LIN {X 0.102,Y -450.857,Z 437.939,A 0.000,B 0.000,C 90.000,E1 204.975} C_DIS
LIN {X -0.124,Y -447.406,Z 437.930,A 0.000,B 0.000,C 90.000,E1 203.387} C_DIS
LIN {X -0.058,Y -442.632,Z 437.917,A 0.000,B 0.000,C 90.000,E1 201.099} C_DIS
LIN {X -0.035,Y -437.484,Z 437.903,A 0.000,B 0.000,C 90.000,E1 198.471} C_DIS
LIN {X 0.091,Y -434.534,Z 437.893,A 0.000,B 0.000,C 90.000,E1 196.804} C_DIS
LIN {X 0.077,Y -430.659,Z 437.881,A 0.000,B 0.000,C 90.000,E1 194.481} C_DIS
LIN {X -0.065,Y -426.530,Z 437.866,A 0.000,B 0.000,C 90.000,E1 191.827} C_DIS
LIN {X -0.012,Y -422.037,Z 437.847,A 0.000,B 0.000,C 90.000,E1 188.454} C_DIS
LIN {X -0.048,Y -419.643,Z 437.836,A 0.000,B 0.000,C 90.000,E1 186.429} C_DIS
LIN {X 0.164,Y -417.753,Z 437.826,A 0.000,B 0.000,C 90.000,E1 184.702} C_DIS
LIN {X -0.025,Y -414.692,Z 437.807,A 0.000,B 0.000,C 90.000,E1 181.318} C_DIS
LIN {X 0.048,Y -412.866,Z 437.792,A 0.000,B 0.000,C 90.000,E1 178.568} C_DIS
LIN {X 0.133,Y -411.529,Z 437.773,A 0.000,B 0.000,C 90.000,E1 175.122} C_DIS
LIN {X -0.070,Y -411.506,Z 437.748,A 0.000,B 0.000,C 90.000,E1 170.679} C_DIS
LIN {X -0.129,Y -412.288,Z 437.733,A 0.000,B 0.000,C 90.000,E1 167.937} C_DIS
LIN {X -0.220,Y -414.218,Z 437.714,A 0.000,B 0.000,C 90.000,E1 164.519} C_DIS
LIN {X 0.137,Y -417.750,Z 437.691,A 0.000,B 0.000,C 90.000,E1 160.369} C_DIS
LIN {X -0.098,Y -422.139,Z 437.670,A 0.000,B 0.000,C 90.000,E1 156.666} C_DIS
LIN {X 0.070,Y -425.355,Z 437.657,A 0.000,B 0.000,C 90.000,E1 154.280} C_DIS
LIN {X 0.108,Y -429.539,Z 437.642,A 0.000,B 0.000,C 90.000,E1 151.591} C_DIS
LIN {X -0.093,Y -432.946,Z 437.631,A 0.000,B 0.000,C 90.000,E1 149.616} C_DIS
LIN {X 0.262,Y -437.222,Z 437.618,A 0.000,B 0.000,C 90.000,E1 147.248} C_DIS
LIN {X -0.031,Y -441.130,Z 437.607,A 0.000,B 0.000,C 90.000,E1 145.308} C_DIS
LIN {X 0.081,Y -447.445,Z 437.591,A 0.000,B 0.000,C 90.000,E1 142.351} C_DIS
LIN {X 0.182,Y -453.544,Z 437.577,A 0.000,B 0.000,C 90.000,E1 139.747} C_DIS
LIN {X 0.005,Y -457.461,Z 437.568,A 0.000,B 0.000,C 90.000,E1 138.162} C_DIS
LIN {X 0.201,Y -461.161,Z 437.559,A 0.000,B 0.000,C 90.000,E1 136.539} C_DIS
LIN {X 0.021,Y -463.308,Z 437.553,A 0.000,B 0.000,C 90.000,E1 135.607} C_DIS
LIN {X -0.141,Y -465.220,Z 437.548,A 0.000,B 0.000,C 90.000,E1 134.676} C_DIS
LIN {X -0.015,Y -466.473,Z 437.545,A 0.000,B 0.000,C 90.000,E1 134.028} C_DIS
LIN {X -0.059,Y -468.597,Z 437.538,A 0.000,B 0.000,C 90.000,E1 132.771} C_DIS
LIN {X -0.151,Y -469.844,Z 437.532,A 0.000,B 0.000,C 90.000,E1 131.838} C_DIS
LIN {X 0.125,Y -470.762,Z 437.527,A 0.000,B 0.000,C 90.000,E1 130.862} C_DIS
LIN {X -0.025,Y -471.260,Z 437.524,A 0.000,B 0.000,C 90.000,E1 130.253} C_DIS
LIN {X -0.096,Y -471.592,Z 437.518,A 0.000,B 0.000,C 90.000,E1 129.322} C_DIS
LIN {X -0.101,Y -471.281,Z 437.513,A 0.000,B 0.000,C 90.000,E1 128.382} C_DIS
LIN {X -0.106,Y -470.509,Z 437.508,A 0.000,B 0.000,C 90.000,E1 127.443} C_DIS
LIN {X -0.119,Y -469.371,Z 437.503,A 0.000,B 0.000,C 90.000,E1 126.503} C_DIS
LIN {X 0.230,Y -467.871,Z 437.498,A 0.000,B 0.000,C 90.000,E1 125.518} C_DIS
LIN {X -0.089,Y -465.949,Z 437.492,A 0.000,B 0.000,C 90.000,E1 124.612} C_DIS
LIN {X -0.041,Y -463.642,Z 437.487,A 0.000,B 0.000,C 90.000,E1 123.658} C_DIS
LIN {X -0.150,Y -461.927,Z 437.483,A 0.000,B 0.000,C 90.000,E1 123.038} C_DIS
LIN {X -0.021,Y -458.176,Z 437.476,A 0.000,B 0.000,C 90.000,E1 121.750} C_DIS
LIN {X 0.043,Y -453.962,Z 437.469,A 0.000,B 0.000,C 90.000,E1 120.463} C_DIS
LIN {X 0.112,Y -450.602,Z 437.464,A 0.000,B 0.000,C 90.000,E1 119.489} C_DIS
LIN {X -0.105,Y -444.709,Z 437.455,A 0.000,B 0.000,C 90.000,E1 117.897} C_DIS
LIN {X -0.140,Y -439.938,Z 437.448,A 0.000,B 0.000,C 90.000,E1 116.616} C_DIS
LIN {X -0.180,Y -439.926,Z 437.448,A 0.000,B 0.000,C 90.000,E1 116.616} C_DIS
LIN {X -0.108,Y -444.759,Z 437.439,A 0.000,B 0.000,C 90.000,E1 114.951} C_DIS
LIN {X -0.138,Y -454.729,Z 437.415,A 0.000,B 0.000,C 90.000,E1 110.737} C_DIS
LIN {X -0.015,Y -457.367,Z 437.410,A 0.000,B 0.000,C 90.000,E1 109.758} C_DIS
LIN {X 0.070,Y -465.999,Z 437.387,A 0.000,B 0.000,C 90.000,E1 105.607} C_DIS
LIN {X -0.207,Y -467.566,Z 437.383,A 0.000,B 0.000,C 90.000,E1 105.009} C_DIS
LIN {X -0.024,Y -468.575,Z 437.380,A 0.000,B 0.000,C 90.000,E1 104.356} C_DIS
LIN {X 0.203,Y -475.799,Z 437.357,A 0.000,B 0.000,C 90.000,E1 100.254} C_DIS
LIN {X 0.041,Y -476.304,Z 437.355,A 0.000,B 0.000,C 90.000,E1 99.962} C_DIS
LIN {X -0.012,Y -481.788,Z 437.331,A 0.000,B 0.000,C 90.000,E1 95.625} C_DIS
LIN {X -0.165,Y -482.171,Z 437.330,A 0.000,B 0.000,C 90.000,E1 95.334} C_DIS
LIN {X -0.235,Y -485.307,Z 437.306,A 0.000,B 0.000,C 90.000,E1 91.031} C_DIS
LIN {X 0.074,Y -485.537,Z 437.304,A 0.000,B 0.000,C 90.000,E1 90.688} C_DIS
LIN {X -0.204,Y -486.319,Z 437.282,A 0.000,B 0.000,C 90.000,E1 86.731} C_DIS
LIN {X -0.069,Y -486.306,Z 437.278,A 0.000,B 0.000,C 90.000,E1 86.102} C_DIS
LIN {X 0.136,Y -484.695,Z 437.254,A 0.000,B 0.000,C 90.000,E1 81.781} C_DIS
LIN {X 0.004,Y -484.601,Z 437.253,A 0.000,B 0.000,C 90.000,E1 81.489} C_DIS
LIN {X -0.116,Y -480.535,Z 437.227,A 0.000,B 0.000,C 90.000,E1 76.881} C_DIS
LIN {X 0.248,Y -474.286,Z 437.201,A 0.000,B 0.000,C 90.000,E1 72.181} C_DIS
LIN {X 0.067,Y -473.850,Z 437.199,A 0.000,B 0.000,C 90.000,E1 71.891} C_DIS
LIN {X 0.175,Y -466.257,Z 437.175,A 0.000,B 0.000,C 90.000,E1 67.486} C_DIS
LIN {X 0.118,Y -465.828,Z 437.173,A 0.000,B 0.000,C 90.000,E1 67.177} C_DIS
LIN {X 0.057,Y -465.235,Z 437.172,A 0.000,B 0.000,C 90.000,E1 66.869} C_DIS
LIN {X -0.019,Y -463.619,Z 437.168,A 0.000,B 0.000,C 90.000,E1 66.177} C_DIS
LIN {X -0.059,Y -463.611,Z 437.168,A 0.000,B 0.000,C 90.000,E1 66.177} C_DIS
LIN {X 0.020,Y -474.649,Z 437.159,A 0.000,B 0.000,C 90.000,E1 64.665} C_DIS
LIN {X -0.068,Y -483.723,Z 437.152,A 0.000,B 0.000,C 90.000,E1 63.435} C_DIS
LIN {X 0.143,Y -487.056,Z 437.150,A 0.000,B 0.000,C 90.000,E1 62.948} C_DIS
LIN {X -0.053,Y -491.221,Z 437.146,A 0.000,B 0.000,C 90.000,E1 62.359} C_DIS
LIN {X 0.047,Y -497.047,Z 437.141,A 0.000,B 0.000,C 90.000,E1 61.435} C_DIS
LIN {X 0.169,Y -501.422,Z 437.137,A 0.000,B 0.000,C 90.000,E1 60.667} C_DIS
LIN {X 0.142,Y -505.295,Z 437.133,A 0.000,B 0.000,C 90.000,E1 59.921} C_DIS
LIN {X 0.082,Y -508.046,Z 437.130,A 0.000,B 0.000,C 90.000,E1 59.331} C_DIS
LIN {X 0.223,Y -509.913,Z 437.127,A 0.000,B 0.000,C 90.000,E1 58.869} C_DIS
LIN {X -0.246,Y -512.107,Z 437.124,A 0.000,B 0.000,C 90.000,E1 58.329} C_DIS
LIN {X 0.095,Y -513.096,Z 437.122,A 0.000,B 0.000,C 90.000,E1 57.995} C_DIS
LIN {X 0.079,Y -514.790,Z 437.119,A 0.000,B 0.000,C 90.000,E1 57.406} C_DIS
LIN {X -0.153,Y -516.775,Z 437.114,A 0.000,B 0.000,C 90.000,E1 56.548} C_DIS
LIN {X 0.141,Y -517.817,Z 437.111,A 0.000,B 0.000,C 90.000,E1 55.928} C_DIS
LIN {X 0.086,Y -518.891,Z 437.106,A 0.000,B 0.000,C 90.000,E1 55.055} C_DIS
LIN {X -0.087,Y -519.451,Z 437.101,A 0.000,B 0.000,C 90.000,E1 54.196} C_DIS
LIN {X 0.165,Y -519.607,Z 437.096,A 0.000,B 0.000,C 90.000,E1 53.290} C_DIS
LIN {X 0.000,Y -519.588,Z 437.091,A 0.000,B 0.000,C 90.000,E1 52.431} C_DIS
LIN {X 0.153,Y -519.326,Z 437.086,A 0.000,B 0.000,C 90.000,E1 51.537} C_DIS
LIN {X 0.251,Y -518.494,Z 437.080,A 0.000,B 0.000,C 90.000,E1 50.356} C_DIS
LIN {X -0.059,Y -517.555,Z 437.073,A 0.000,B 0.000,C 90.000,E1 49.218} C_DIS
LIN {X 0.003,Y -516.367,Z 437.067,A 0.000,B 0.000,C 90.000,E1 48.038} C_DIS
LIN {X -0.106,Y -514.780,Z 437.059,A 0.000,B 0.000,C 90.000,E1 46.581} C_DIS
LIN {X -0.276,Y -511.804,Z 437.044,A 0.000,B 0.000,C 90.000,E1 43.947} C_DIS
LIN {X -0.091,Y -510.209,Z 437.036,A 0.000,B 0.000,C 90.000,E1 42.447} C_DIS
LIN {X 0.200,Y -509.021,Z 437.029,A 0.000,B 0.000,C 90.000,E1 41.229} C_DIS
LIN {X -0.101,Y -506.220,Z 437.014,A 0.000,B 0.000,C 90.000,E1 38.588} C_DIS
LIN {X 0.091,Y -504.707,Z 437.006,A 0.000,B 0.000,C 90.000,E1 37.076} C_DIS
LIN {X 0.176,Y -503.686,Z 437.001,A 0.000,B 0.000,C 90.000,E1 36.171} C_DIS
LIN {X 0.029,Y -501.970,Z 436.993,A 0.000,B 0.000,C 90.000,E1 34.692} C_DIS
LIN {X 0.259,Y -500.091,Z 436.984,A 0.000,B 0.000,C 90.000,E1 33.166} C_DIS
LIN {X 0.064,Y -497.370,Z 436.973,A 0.000,B 0.000,C 90.000,E1 31.082} C_DIS
LIN {X -0.078,Y -495.355,Z 436.964,A 0.000,B 0.000,C 90.000,E1 29.589} C_DIS
LIN {X 0.228,Y -492.204,Z 436.951,A 0.000,B 0.000,C 90.000,E1 27.129} C_DIS
LIN {X 0.267,Y -488.755,Z 436.934,A 0.000,B 0.000,C 90.000,E1 24.079} C_DIS
LIN {X 0.006,Y -486.549,Z 436.920,A 0.000,B 0.000,C 90.000,E1 21.663} C_DIS
LIN {X 0.105,Y -485.254,Z 436.910,A 0.000,B 0.000,C 90.000,E1 19.812} C_DIS
LIN {X -0.156,Y -483.886,Z 436.898,A 0.000,B 0.000,C 90.000,E1 17.692} C_DIS
LIN {X 0.158,Y -483.262,Z 436.893,A 0.000,B 0.000,C 90.000,E1 16.732} C_DIS
LIN {X 0.036,Y -481.976,Z 436.883,A 0.000,B 0.000,C 90.000,E1 14.898} C_DIS
LIN {X 0.223,Y -480.003,Z 436.864,A 0.000,B 0.000,C 90.000,E1 11.478} C_DIS
LIN {X -0.002,Y -479.129,Z 436.850,A 0.000,B 0.000,C 90.000,E1 9.029} C_DIS
LIN {X -0.150,Y -478.666,Z 436.835,A 0.000,B 0.000,C 90.000,E1 6.258} C_DIS
LIN {X -0.195,Y -478.900,Z 436.821,A 0.000,B 0.000,C 90.000,E1 3.784} C_DIS
LIN {X -0.110,Y -480.493,Z 436.800,A 0.000,B 0.000,C 90.000,E1 0.057} C_DIS
LIN {X -0.097,Y -481.532,Z 436.792,A 0.000,B 0.000,C 90.000,E1 358.568} C_DIS
LIN {X -0.057,Y -483.080,Z 436.783,A 0.000,B 0.000,C 90.000,E1 357.020} C_DIS
LIN {X -0.092,Y -487.702,Z 436.763,A 0.000,B 0.000,C 90.000,E1 353.337} C_DIS
LIN {X -0.004,Y -492.402,Z 436.746,A 0.000,B 0.000,C 90.000,E1 350.274} C_DIS
LIN {X 0.038,Y -498.428,Z 436.728,A 0.000,B 0.000,C 90.000,E1 346.937} C_DIS
LIN {X 0.083,Y -505.796,Z 436.709,A 0.000,B 0.000,C 90.000,E1 343.630} C_DIS
LIN {X -0.024,Y -512.499,Z 436.694,A 0.000,B 0.000,C 90.000,E1 340.967} C_DIS
LIN {X 0.004,Y -518.050,Z 436.683,A 0.000,B 0.000,C 90.000,E1 338.901} C_DIS
LIN {X -0.086,Y -522.817,Z 436.673,A 0.000,B 0.000,C 90.000,E1 337.155} C_DIS
LIN {X 0.245,Y -526.906,Z 436.665,A 0.000,B 0.000,C 90.000,E1 335.665} C_DIS
LIN {X 0.275,Y -532.592,Z 436.654,A 0.000,B 0.000,C 90.000,E1 333.640} C_DIS
LIN {X 0.207,Y -538.348,Z 436.643,A 0.000,B 0.000,C 90.000,E1 331.641} C_DIS
LIN {X 0.058,Y -543.469,Z 436.633,A 0.000,B 0.000,C 90.000,E1 329.950} C_DIS
LIN {X 0.065,Y -547.624,Z 436.625,A 0.000,B 0.000,C 90.000,E1 328.535} C_DIS
LIN {X 0.103,Y -550.994,Z 436.619,A 0.000,B 0.000,C 90.000,E1 327.406} C_DIS
LIN {X -0.013,Y -557.487,Z 436.607,A 0.000,B 0.000,C 90.000,E1 325.182} C_DIS
LIN {X 0.186,Y -562.446,Z 436.597,A 0.000,B 0.000,C 90.000,E1 323.497} C_DIS
LIN {X 0.266,Y -566.630,Z 436.590,A 0.000,B 0.000,C 90.000,E1 322.110} C_DIS
LIN {X 0.381,Y -573.652,Z 436.578,A 0.000,B 0.000,C 90.000,E1 319.908} C_DIS
LIN {X 0.078,Y -579.838,Z 436.567,A 0.000,B 0.000,C 90.000,E1 318.038} C_DIS
LIN {X -0.301,Y -584.991,Z 436.558,A 0.000,B 0.000,C 90.000,E1 316.458} C_DIS
LIN {X 0.089,Y -589.319,Z 436.551,A 0.000,B 0.000,C 90.000,E1 315.081} C_DIS
LIN {X -0.280,Y -593.754,Z 436.543,A 0.000,B 0.000,C 90.000,E1 313.785} C_DIS
LIN {X 0.073,Y -599.031,Z 436.534,A 0.000,B 0.000,C 90.000,E1 312.162} C_DIS
LIN {X -0.311,Y -604.180,Z 436.526,A 0.000,B 0.000,C 90.000,E1 310.620} C_DIS
LIN {X -0.143,Y -609.193,Z 436.517,A 0.000,B 0.000,C 90.000,E1 309.036} C_DIS
LIN {X -0.166,Y -611.630,Z 436.513,A 0.000,B 0.000,C 90.000,E1 308.257} C_DIS
LIN {X 0.254,Y -616.294,Z 436.504,A 0.000,B 0.000,C 90.000,E1 306.664} C_DIS
LIN {X 0.083,Y -620.071,Z 436.497,A 0.000,B 0.000,C 90.000,E1 305.391} C_DIS
LIN {X -0.358,Y -623.004,Z 436.491,A 0.000,B 0.000,C 90.000,E1 304.405} C_DIS
LIN {X 0.083,Y -627.210,Z 436.482,A 0.000,B 0.000,C 90.000,E1 302.832} C_DIS
LIN {X -0.257,Y -631.166,Z 436.474,A 0.000,B 0.000,C 90.000,E1 301.337} C_DIS
LIN {X -0.025,Y -634.326,Z 436.467,A 0.000,B 0.000,C 90.000,E1 300.050} C_DIS
LIN {X 0.136,Y -636.758,Z 436.461,A 0.000,B 0.000,C 90.000,E1 299.027} C_DIS
LIN {X 0.197,Y -640.277,Z 436.453,A 0.000,B 0.000,C 90.000,E1 297.513} C_DIS
LIN {X -0.054,Y -643.084,Z 436.446,A 0.000,B 0.000,C 90.000,E1 296.283} C_DIS
LIN {X -0.118,Y -644.697,Z 436.442,A 0.000,B 0.000,C 90.000,E1 295.540} C_DIS
LIN {X 0.094,Y -647.710,Z 436.434,A 0.000,B 0.000,C 90.000,E1 294.027} C_DIS
LIN {X 0.181,Y -649.526,Z 436.428,A 0.000,B 0.000,C 90.000,E1 293.025} C_DIS
LIN {X 0.136,Y -651.609,Z 436.421,A 0.000,B 0.000,C 90.000,E1 291.791} C_DIS
LIN {X 0.124,Y -653.574,Z 436.414,A 0.000,B 0.000,C 90.000,E1 290.556} C_DIS
LIN {X 0.041,Y -655.143,Z 436.409,A 0.000,B 0.000,C 90.000,E1 289.577} C_DIS
LIN {X -0.267,Y -656.953,Z 436.401,A 0.000,B 0.000,C 90.000,E1 288.127} C_DIS
LIN {X 0.193,Y -658.141,Z 436.394,A 0.000,B 0.000,C 90.000,E1 286.858} C_DIS
LIN {X -0.157,Y -659.115,Z 436.387,A 0.000,B 0.000,C 90.000,E1 285.662} C_DIS
LIN {X 0.072,Y -659.717,Z 436.382,A 0.000,B 0.000,C 90.000,E1 284.662} C_DIS
LIN {X 0.374,Y -660.314,Z 436.375,A 0.000,B 0.000,C 90.000,E1 283.411} C_DIS
LIN {X -0.169,Y -660.599,Z 436.369,A 0.000,B 0.000,C 90.000,E1 282.479} C_DIS
LIN {X -0.018,Y -660.661,Z 436.362,A 0.000,B 0.000,C 90.000,E1 281.243} C_DIS
LIN {X 0.099,Y -660.617,Z 436.357,A 0.000,B 0.000,C 90.000,E1 280.254} C_DIS
LIN {X 0.218,Y -660.279,Z 436.352,A 0.000,B 0.000,C 90.000,E1 279.265} C_DIS
LIN {X 0.326,Y -659.859,Z 436.346,A 0.000,B 0.000,C 90.000,E1 278.276} C_DIS
LIN {X 0.130,Y -659.052,Z 436.339,A 0.000,B 0.000,C 90.000,E1 277.068} C_DIS
LIN {X 0.134,Y -658.133,Z 436.334,A 0.000,B 0.000,C 90.000,E1 276.087} C_DIS
LIN {X -0.075,Y -656.630,Z 436.327,A 0.000,B 0.000,C 90.000,E1 274.878} C_DIS
LIN {X -0.316,Y -654.805,Z 436.320,A 0.000,B 0.000,C 90.000,E1 273.669} C_DIS
LIN {X 0.020,Y -652.674,Z 436.313,A 0.000,B 0.000,C 90.000,E1 272.407} C_DIS
LIN {X -0.125,Y -650.827,Z 436.308,A 0.000,B 0.000,C 90.000,E1 271.432} C_DIS
LIN {X -0.312,Y -648.778,Z 436.302,A 0.000,B 0.000,C 90.000,E1 270.458} C_DIS
LIN {X -0.095,Y -645.959,Z 436.296,A 0.000,B 0.000,C 90.000,E1 269.198} C_DIS
LIN {X 0.295,Y -643.507,Z 436.290,A 0.000,B 0.000,C 90.000,E1 268.167} C_DIS
LIN {X -0.211,Y -640.249,Z 436.283,A 0.000,B 0.000,C 90.000,E1 266.963} C_DIS
LIN {X 0.293,Y -636.092,Z 436.275,A 0.000,B 0.000,C 90.000,E1 265.412} C_DIS
LIN {X -0.280,Y -632.652,Z 436.268,A 0.000,B 0.000,C 90.000,E1 264.204} C_DIS
LIN {X -0.207,Y -629.005,Z 436.261,A 0.000,B 0.000,C 90.000,E1 262.932} C_DIS
LIN {X -0.188,Y -625.295,Z 436.254,A 0.000,B 0.000,C 90.000,E1 261.659} C_DIS
LIN {X -0.237,Y -621.464,Z 436.247,A 0.000,B 0.000,C 90.000,E1 260.387} C_DIS
LIN {X 0.123,Y -616.805,Z 436.238,A 0.000,B 0.000,C 90.000,E1 258.814} C_DIS
LIN {X -0.211,Y -613.555,Z 436.232,A 0.000,B 0.000,C 90.000,E1 257.813} C_DIS
LIN {X 0.017,Y -610.264,Z 436.226,A 0.000,B 0.000,C 90.000,E1 256.756} C_DIS
LIN {X -0.067,Y -606.024,Z 436.219,A 0.000,B 0.000,C 90.000,E1 255.463} C_DIS
LIN {X 0.226,Y -600.736,Z 436.211,A 0.000,B 0.000,C 90.000,E1 253.866} C_DIS
LIN {X 0.290,Y -596.217,Z 436.203,A 0.000,B 0.000,C 90.000,E1 252.543} C_DIS
LIN {X -0.283,Y -591.619,Z 436.196,A 0.000,B 0.000,C 90.000,E1 251.275} C_DIS
LIN {X -0.176,Y -586.888,Z 436.188,A 0.000,B 0.000,C 90.000,E1 249.934} C_DIS
LIN {X -0.017,Y -583.015,Z 436.183,A 0.000,B 0.000,C 90.000,E1 248.847} C_DIS
LIN {X 0.139,Y -577.959,Z 436.175,A 0.000,B 0.000,C 90.000,E1 247.486} C_DIS
LIN {X 0.066,Y -573.770,Z 436.169,A 0.000,B 0.000,C 90.000,E1 246.410} C_DIS
LIN {X 0.056,Y -568.414,Z 436.161,A 0.000,B 0.000,C 90.000,E1 245.049} C_DIS
LIN {X -0.083,Y -562.965,Z 436.154,A 0.000,B 0.000,C 90.000,E1 243.691} C_DIS
LIN {X 0.195,Y -557.542,Z 436.146,A 0.000,B 0.000,C 90.000,E1 242.281} C_DIS
LIN {X 0.170,Y -550.030,Z 436.135,A 0.000,B 0.000,C 90.000,E1 240.333} C_DIS
LIN {X 0.009,Y -543.724,Z 436.126,A 0.000,B 0.000,C 90.000,E1 238.663} C_DIS
LIN {X -0.007,Y -538.580,Z 436.118,A 0.000,B 0.000,C 90.000,E1 237.248} C_DIS
LIN {X 0.174,Y -533.391,Z 436.110,A 0.000,B 0.000,C 90.000,E1 235.801} C_DIS
LIN {X 0.179,Y -525.251,Z 436.097,A 0.000,B 0.000,C 90.000,E1 233.497} C_DIS
LIN {X -0.062,Y -519.255,Z 436.088,A 0.000,B 0.000,C 90.000,E1 231.778} C_DIS
LIN {X -0.029,Y -508.135,Z 436.068,A 0.000,B 0.000,C 90.000,E1 228.243} C_DIS
LIN {X -0.045,Y -502.925,Z 436.058,A 0.000,B 0.000,C 90.000,E1 226.458} C_DIS
LIN {X -0.189,Y -497.877,Z 436.048,A 0.000,B 0.000,C 90.000,E1 224.676} C_DIS
LIN {X 0.090,Y -492.012,Z 436.036,A 0.000,B 0.000,C 90.000,E1 222.528} C_DIS
LIN {X 0.255,Y -487.958,Z 436.028,A 0.000,B 0.000,C 90.000,E1 220.987} C_DIS
LIN {X -0.032,Y -482.459,Z 436.016,A 0.000,B 0.000,C 90.000,E1 218.874} C_DIS
LIN {X 0.089,Y -478.635,Z 436.007,A 0.000,B 0.000,C 90.000,E1 217.317} C_DIS
LIN {X 0.185,Y -472.858,Z 435.994,A 0.000,B 0.000,C 90.000,E1 214.818} C_DIS
LIN {X 0.024,Y -468.678,Z 435.983,A 0.000,B 0.000,C 90.000,E1 212.959} C_DIS
LIN {X -0.140,Y -465.976,Z 435.976,A 0.000,B 0.000,C 90.000,E1 211.720} C_DIS
LIN {X 0.081,Y -461.920,Z 435.966,A 0.000,B 0.000,C 90.000,E1 209.795} C_DIS
LIN {X -0.133,Y -458.570,Z 435.957,A 0.000,B 0.000,C 90.000,E1 208.231} C_DIS
LIN {X -0.006,Y -455.180,Z 435.948,A 0.000,B 0.000,C 90.000,E1 206.616} C_DIS
LIN {X -0.148,Y -451.748,Z 435.939,A 0.000,B 0.000,C 90.000,E1 205.027} C_DIS
LIN {X 0.052,Y -448.270,Z 435.930,A 0.000,B 0.000,C 90.000,E1 203.387} C_DIS
LIN {X 0.138,Y -443.442,Z 435.917,A 0.000,B 0.000,C 90.000,E1 201.099} C_DIS
LIN {X 0.045,Y -438.249,Z 435.903,A 0.000,B 0.000,C 90.000,E1 198.489} C_DIS
LIN {X -0.093,Y -435.274,Z 435.894,A 0.000,B 0.000,C 90.000,E1 196.858} C_DIS
LIN {X -0.090,Y -431.379,Z 435.881,A 0.000,B 0.000,C 90.000,E1 194.537} C_DIS
LIN {X 0.205,Y -427.197,Z 435.866,A 0.000,B 0.000,C 90.000,E1 191.827} C_DIS
LIN {X -0.136,Y -422.697,Z 435.847,A 0.000,B 0.000,C 90.000,E1 188.511} C_DIS
LIN {X -0.137,Y -419.901,Z 435.834,A 0.000,B 0.000,C 90.000,E1 186.144} C_DIS
LIN {X -0.163,Y -416.128,Z 435.813,A 0.000,B 0.000,C 90.000,E1 182.407} C_DIS
LIN {X -0.014,Y -413.673,Z 435.794,A 0.000,B 0.000,C 90.000,E1 178.969} C_DIS
LIN {X 0.104,Y -412.121,Z 435.773,A 0.000,B 0.000,C 90.000,E1 175.179} C_DIS
LIN {X -0.030,Y -412.135,Z 435.747,A 0.000,B 0.000,C 90.000,E1 170.387} C_DIS
LIN {X -0.102,Y -412.842,Z 435.733,A 0.000,B 0.000,C 90.000,E1 167.993} C_DIS
LIN {X -0.022,Y -415.002,Z 435.712,A 0.000,B 0.000,C 90.000,E1 164.212} C_DIS
LIN {X 0.228,Y -418.330,Z 435.691,A 0.000,B 0.000,C 90.000,E1 160.423} C_DIS
LIN {X -0.132,Y -420.137,Z 435.682,A 0.000,B 0.000,C 90.000,E1 158.773} C_DIS
LIN {X 0.201,Y -423.169,Z 435.669,A 0.000,B 0.000,C 90.000,E1 156.357} C_DIS
LIN {X 0.013,Y -426.461,Z 435.656,A 0.000,B 0.000,C 90.000,E1 154.024} C_DIS
LIN {X -0.086,Y -430.185,Z 435.643,A 0.000,B 0.000,C 90.000,E1 151.691} C_DIS
LIN {X 0.130,Y -434.229,Z 435.630,A 0.000,B 0.000,C 90.000,E1 149.331} C_DIS
LIN {X -0.132,Y -437.347,Z 435.621,A 0.000,B 0.000,C 90.000,E1 147.709} C_DIS
LIN {X -0.013,Y -441.987,Z 435.608,A 0.000,B 0.000,C 90.000,E1 145.388} C_DIS
LIN {X 0.072,Y -447.640,Z 435.593,A 0.000,B 0.000,C 90.000,E1 142.763} C_DIS
LIN {X -0.154,Y -451.477,Z 435.584,A 0.000,B 0.000,C 90.000,E1 141.170} C_DIS
LIN {X -0.028,Y -455.414,Z 435.575,A 0.000,B 0.000,C 90.000,E1 139.542} C_DIS
LIN {X 0.131,Y -459.422,Z 435.566,A 0.000,B 0.000,C 90.000,E1 137.919} C_DIS
LIN {X 0.035,Y -463.193,Z 435.557,A 0.000,B 0.000,C 90.000,E1 136.338} C_DIS
LIN {X -0.056,Y -465.989,Z 435.550,A 0.000,B 0.000,C 90.000,E1 135.081} C_DIS
LIN {X 0.218,Y -468.517,Z 435.543,A 0.000,B 0.000,C 90.000,E1 133.785} C_DIS
LIN {X 0.205,Y -470.655,Z 435.536,A 0.000,B 0.000,C 90.000,E1 132.528} C_DIS
LIN {X 0.136,Y -471.837,Z 435.531,A 0.000,B 0.000,C 90.000,E1 131.595} C_DIS
LIN {X -0.008,Y -472.515,Z 435.528,A 0.000,B 0.000,C 90.000,E1 130.987} C_DIS
LIN {X 0.298,Y -473.225,Z 435.523,A 0.000,B 0.000,C 90.000,E1 130.011} C_DIS
LIN {X -0.054,Y -473.512,Z 435.517,A 0.000,B 0.000,C 90.000,E1 129.116} C_DIS
LIN {X -0.034,Y -473.134,Z 435.512,A 0.000,B 0.000,C 90.000,E1 128.177} C_DIS
LIN {X -0.015,Y -472.302,Z 435.507,A 0.000,B 0.000,C 90.000,E1 127.237} C_DIS
LIN {X -0.008,Y -471.086,Z 435.502,A 0.000,B 0.000,C 90.000,E1 126.297} C_DIS
LIN {X -0.019,Y -469.565,Z 435.496,A 0.000,B 0.000,C 90.000,E1 125.358} C_DIS
LIN {X -0.091,Y -468.273,Z 435.493,A 0.000,B 0.000,C 90.000,E1 124.739} C_DIS
LIN {X -0.019,Y -465.974,Z 435.488,A 0.000,B 0.000,C 90.000,E1 123.785} C_DIS
LIN {X -0.113,Y -464.354,Z 435.484,A 0.000,B 0.000,C 90.000,E1 123.166} C_DIS
LIN {X 0.051,Y -460.561,Z 435.477,A 0.000,B 0.000,C 90.000,E1 121.878} C_DIS
LIN {X 0.035,Y -457.455,Z 435.472,A 0.000,B 0.000,C 90.000,E1 120.924} C_DIS
LIN {X -0.252,Y -454.107,Z 435.467,A 0.000,B 0.000,C 90.000,E1 120.001} C_DIS
LIN {X 0.042,Y -450.609,Z 435.461,A 0.000,B 0.000,C 90.000,E1 118.999} C_DIS
LIN {X -0.067,Y -445.815,Z 435.454,A 0.000,B 0.000,C 90.000,E1 117.719} C_DIS
LIN {X 0.031,Y -441.501,Z 435.448,A 0.000,B 0.000,C 90.000,E1 116.565} C_DIS
LIN {X -0.044,Y -440.628,Z 435.446,A 0.000,B 0.000,C 90.000,E1 116.360} C_DIS
LIN {X -0.084,Y -440.609,Z 435.446,A 0.000,B 0.000,C 90.000,E1 116.360} C_DIS
LIN {X 0.117,Y -444.288,Z 435.439,A 0.000,B 0.000,C 90.000,E1 115.079} C_DIS
LIN {X -0.030,Y -445.135,Z 435.438,A 0.000,B 0.000,C 90.000,E1 114.771} C_DIS
LIN {X 0.076,Y -454.312,Z 435.416,A 0.000,B 0.000,C 90.000,E1 110.865} C_DIS
LIN {X -0.232,Y -456.979,Z 435.411,A 0.000,B 0.000,C 90.000,E1 109.939} C_DIS
LIN {X 0.006,Y -458.242,Z 435.407,A 0.000,B 0.000,C 90.000,E1 109.268} C_DIS
LIN {X 0.204,Y -466.400,Z 435.386,A 0.000,B 0.000,C 90.000,E1 105.426} C_DIS
LIN {X -0.072,Y -467.914,Z 435.382,A 0.000,B 0.000,C 90.000,E1 104.828} C_DIS
LIN {X -0.045,Y -475.486,Z 435.358,A 0.000,B 0.000,C 90.000,E1 100.433} C_DIS
LIN {X -0.206,Y -476.130,Z 435.356,A 0.000,B 0.000,C 90.000,E1 100.141} C_DIS
LIN {X 0.076,Y -482.044,Z 435.330,A 0.000,B 0.000,C 90.000,E1 95.454} C_DIS
LIN {X -0.133,Y -485.477,Z 435.305,A 0.000,B 0.000,C 90.000,E1 90.859} C_DIS
LIN {X 0.074,Y -486.247,Z 435.283,A 0.000,B 0.000,C 90.000,E1 86.846} C_DIS
LIN {X -0.100,Y -486.386,Z 435.281,A 0.000,B 0.000,C 90.000,E1 86.560} C_DIS
LIN {X 0.210,Y -486.363,Z 435.279,A 0.000,B 0.000,C 90.000,E1 86.216} C_DIS
LIN {X -0.187,Y -484.690,Z 435.254,A 0.000,B 0.000,C 90.000,E1 81.659} C_DIS
LIN {X -0.172,Y -483.692,Z 435.248,A 0.000,B 0.000,C 90.000,E1 80.735} C_DIS
LIN {X 0.191,Y -480.624,Z 435.228,A 0.000,B 0.000,C 90.000,E1 76.992} C_DIS
LIN {X 0.050,Y -480.300,Z 435.226,A 0.000,B 0.000,C 90.000,E1 76.700} C_DIS
LIN {X -0.046,Y -474.120,Z 435.200,A 0.000,B 0.000,C 90.000,E1 72.054} C_DIS
LIN {X -0.178,Y -465.584,Z 435.172,A 0.000,B 0.000,C 90.000,E1 67.050} C_DIS
LIN {X 0.191,Y -464.085,Z 435.169,A 0.000,B 0.000,C 90.000,E1 66.357} C_DIS
LIN {X 0.151,Y -464.104,Z 435.169,A 0.000,B 0.000,C 90.000,E1 66.357} C_DIS
LIN {X -0.080,Y -474.200,Z 435.161,A 0.000,B 0.000,C 90.000,E1 65.025} C_DIS
LIN {X 0.247,Y -482.201,Z 435.155,A 0.000,B 0.000,C 90.000,E1 63.896} C_DIS
LIN {X 0.238,Y -487.857,Z 435.151,A 0.000,B 0.000,C 90.000,E1 63.127} C_DIS
LIN {X 0.050,Y -492.060,Z 435.148,A 0.000,B 0.000,C 90.000,E1 62.538} C_DIS
LIN {X 0.129,Y -496.938,Z 435.143,A 0.000,B 0.000,C 90.000,E1 61.769} C_DIS
LIN {X 0.206,Y -499.713,Z 435.141,A 0.000,B 0.000,C 90.000,E1 61.307} C_DIS
LIN {X 0.108,Y -503.106,Z 435.137,A 0.000,B 0.000,C 90.000,E1 60.717} C_DIS
LIN {X 0.095,Y -507.682,Z 435.132,A 0.000,B 0.000,C 90.000,E1 59.822} C_DIS
LIN {X -0.131,Y -510.346,Z 435.129,A 0.000,B 0.000,C 90.000,E1 59.253} C_DIS
LIN {X 0.024,Y -512.146,Z 435.127,A 0.000,B 0.000,C 90.000,E1 58.791} C_DIS
LIN {X 0.006,Y -514.281,Z 435.123,A 0.000,B 0.000,C 90.000,E1 58.201} C_DIS
LIN {X -0.079,Y -516.713,Z 435.118,A 0.000,B 0.000,C 90.000,E1 57.327} C_DIS
LIN {X 0.210,Y -518.076,Z 435.115,A 0.000,B 0.000,C 90.000,E1 56.707} C_DIS
LIN {X -0.271,Y -519.539,Z 435.110,A 0.000,B 0.000,C 90.000,E1 55.881} C_DIS
LIN {X 0.042,Y -520.256,Z 435.107,A 0.000,B 0.000,C 90.000,E1 55.261} C_DIS
LIN {X -0.117,Y -520.892,Z 435.102,A 0.000,B 0.000,C 90.000,E1 54.402} C_DIS
LIN {X 0.155,Y -521.122,Z 435.097,A 0.000,B 0.000,C 90.000,E1 53.497} C_DIS
LIN {X 0.006,Y -521.081,Z 435.092,A 0.000,B 0.000,C 90.000,E1 52.637} C_DIS
LIN {X 0.178,Y -520.824,Z 435.088,A 0.000,B 0.000,C 90.000,E1 51.743} C_DIS
LIN {X -0.028,Y -520.007,Z 435.081,A 0.000,B 0.000,C 90.000,E1 50.598} C_DIS
LIN {X -0.322,Y -519.050,Z 435.075,A 0.000,B 0.000,C 90.000,E1 49.461} C_DIS
LIN {X 0.106,Y -517.840,Z 435.068,A 0.000,B 0.000,C 90.000,E1 48.243} C_DIS
LIN {X 0.051,Y -516.187,Z 435.060,A 0.000,B 0.000,C 90.000,E1 46.782} C_DIS
LIN {X -0.248,Y -513.724,Z 435.049,A 0.000,B 0.000,C 90.000,E1 44.757} C_DIS
LIN {X -0.022,Y -512.154,Z 435.040,A 0.000,B 0.000,C 90.000,E1 43.257} C_DIS
LIN {X 0.320,Y -509.962,Z 435.029,A 0.000,B 0.000,C 90.000,E1 41.148} C_DIS
LIN {X -0.172,Y -507.478,Z 435.016,A 0.000,B 0.000,C 90.000,E1 38.830} C_DIS
LIN {X 0.051,Y -505.928,Z 435.007,A 0.000,B 0.000,C 90.000,E1 37.317} C_DIS
LIN {X -0.060,Y -504.552,Z 435.001,A 0.000,B 0.000,C 90.000,E1 36.137} C_DIS
LIN {X 0.213,Y -502.826,Z 434.992,A 0.000,B 0.000,C 90.000,E1 34.612} C_DIS
LIN {X -0.238,Y -500.937,Z 434.984,A 0.000,B 0.000,C 90.000,E1 33.166} C_DIS
LIN {X -0.152,Y -498.203,Z 434.972,A 0.000,B 0.000,C 90.000,E1 31.052} C_DIS
LIN {X -0.102,Y -496.197,Z 434.964,A 0.000,B 0.000,C 90.000,E1 29.539} C_DIS
LIN {X -0.199,Y -493.037,Z 434.951,A 0.000,B 0.000,C 90.000,E1 27.129} C_DIS
LIN {X -0.153,Y -489.928,Z 434.935,A 0.000,B 0.000,C 90.000,E1 24.387} C_DIS
LIN {X 0.253,Y -487.656,Z 434.922,A 0.000,B 0.000,C 90.000,E1 21.897} C_DIS
LIN {X 0.202,Y -486.339,Z 434.912,A 0.000,B 0.000,C 90.000,E1 20.066} C_DIS
LIN {X -0.021,Y -484.953,Z 434.900,A 0.000,B 0.000,C 90.000,E1 17.946} C_DIS
LIN {X -0.151,Y -484.121,Z 434.893,A 0.000,B 0.000,C 90.000,E1 16.732} C_DIS
LIN {X -0.129,Y -482.817,Z 434.883,A 0.000,B 0.000,C 90.000,E1 14.883} C_DIS
LIN {X 0.110,Y -480.999,Z 434.866,A 0.000,B 0.000,C 90.000,E1 11.771} C_DIS
LIN {X 0.063,Y -480.190,Z 434.853,A 0.000,B 0.000,C 90.000,E1 9.613} C_DIS
LIN {X -0.093,Y -479.665,Z 434.841,A 0.000,B 0.000,C 90.000,E1 7.466} C_DIS
LIN {X -0.165,Y -479.725,Z 434.823,A 0.000,B 0.000,C 90.000,E1 4.069} C_DIS
LIN {X -0.049,Y -481.236,Z 434.802,A 0.000,B 0.000,C 90.000,E1 0.344} C_DIS
LIN {X -0.083,Y -482.496,Z 434.792,A 0.000,B 0.000,C 90.000,E1 358.568} C_DIS
LIN {X 0.120,Y -484.688,Z 434.780,A 0.000,B 0.000,C 90.000,E1 356.388} C_DIS
LIN {X -0.195,Y -487.776,Z 434.766,A 0.000,B 0.000,C 90.000,E1 353.970} C_DIS
LIN {X -0.248,Y -490.903,Z 434.755,A 0.000,B 0.000,C 90.000,E1 351.837} C_DIS
LIN {X 0.111,Y -493.397,Z 434.746,A 0.000,B 0.000,C 90.000,E1 350.274} C_DIS
LIN {X -0.235,Y -498.245,Z 434.731,A 0.000,B 0.000,C 90.000,E1 347.589} C_DIS
LIN {X -0.073,Y -503.992,Z 434.716,A 0.000,B 0.000,C 90.000,E1 344.866} C_DIS
LIN {X -0.180,Y -508.266,Z 434.706,A 0.000,B 0.000,C 90.000,E1 343.087} C_DIS
LIN {X 0.165,Y -514.318,Z 434.693,A 0.000,B 0.000,C 90.000,E1 340.678} C_DIS
LIN {X -0.066,Y -519.873,Z 434.681,A 0.000,B 0.000,C 90.000,E1 338.646} C_DIS
LIN {X -0.155,Y -525.541,Z 434.670,A 0.000,B 0.000,C 90.000,E1 336.613} C_DIS
LIN {X -0.045,Y -529.574,Z 434.662,A 0.000,B 0.000,C 90.000,E1 335.153} C_DIS
LIN {X -0.139,Y -534.524,Z 434.652,A 0.000,B 0.000,C 90.000,E1 333.435} C_DIS
LIN {X -0.140,Y -539.478,Z 434.643,A 0.000,B 0.000,C 90.000,E1 331.719} C_DIS
LIN {X -0.002,Y -544.628,Z 434.633,A 0.000,B 0.000,C 90.000,E1 329.999} C_DIS
LIN {X -0.002,Y -548.008,Z 434.627,A 0.000,B 0.000,C 90.000,E1 328.869} C_DIS
LIN {X 0.092,Y -552.215,Z 434.619,A 0.000,B 0.000,C 90.000,E1 327.454} C_DIS
LIN {X -0.057,Y -557.937,Z 434.608,A 0.000,B 0.000,C 90.000,E1 325.515} C_DIS
LIN {X -0.073,Y -563.777,Z 434.598,A 0.000,B 0.000,C 90.000,E1 323.577} C_DIS
LIN {X 0.146,Y -568.807,Z 434.589,A 0.000,B 0.000,C 90.000,E1 321.904} C_DIS
LIN {X -0.126,Y -575.873,Z 434.576,A 0.000,B 0.000,C 90.000,E1 319.747} C_DIS
LIN {X 0.287,Y -581.184,Z 434.567,A 0.000,B 0.000,C 90.000,E1 318.081} C_DIS
LIN {X -0.051,Y -586.388,Z 434.558,A 0.000,B 0.000,C 90.000,E1 316.500} C_DIS
LIN {X -0.042,Y -590.801,Z 434.551,A 0.000,B 0.000,C 90.000,E1 315.162} C_DIS
LIN {X 0.227,Y -596.105,Z 434.542,A 0.000,B 0.000,C 90.000,E1 313.542} C_DIS
LIN {X -0.217,Y -601.409,Z 434.533,A 0.000,B 0.000,C 90.000,E1 312.000} C_DIS
LIN {X 0.040,Y -605.725,Z 434.526,A 0.000,B 0.000,C 90.000,E1 310.663} C_DIS
LIN {X 0.043,Y -609.951,Z 434.519,A 0.000,B 0.000,C 90.000,E1 309.358} C_DIS
LIN {X 0.222,Y -613.205,Z 434.513,A 0.000,B 0.000,C 90.000,E1 308.302} C_DIS
LIN {X -0.195,Y -617.952,Z 434.504,A 0.000,B 0.000,C 90.000,E1 306.790} C_DIS
LIN {X -0.346,Y -621.710,Z 434.497,A 0.000,B 0.000,C 90.000,E1 305.518} C_DIS
LIN {X 0.078,Y -625.404,Z 434.490,A 0.000,B 0.000,C 90.000,E1 304.199} C_DIS
LIN {X -0.303,Y -628.936,Z 434.483,A 0.000,B 0.000,C 90.000,E1 302.959} C_DIS
LIN {X -0.076,Y -632.948,Z 434.475,A 0.000,B 0.000,C 90.000,E1 301.416} C_DIS
LIN {X 0.156,Y -635.507,Z 434.469,A 0.000,B 0.000,C 90.000,E1 300.384} C_DIS
LIN {X -0.175,Y -638.603,Z 434.462,A 0.000,B 0.000,C 90.000,E1 299.155} C_DIS
LIN {X -0.079,Y -642.149,Z 434.454,A 0.000,B 0.000,C 90.000,E1 297.641} C_DIS
LIN {X 0.356,Y -645.521,Z 434.445,A 0.000,B 0.000,C 90.000,E1 296.104} C_DIS
LIN {X -0.264,Y -647.143,Z 434.441,A 0.000,B 0.000,C 90.000,E1 295.412} C_DIS
LIN {X 0.170,Y -649.686,Z 434.434,A 0.000,B 0.000,C 90.000,E1 294.131} C_DIS
LIN {X 0.018,Y -651.495,Z 434.429,A 0.000,B 0.000,C 90.000,E1 293.153} C_DIS
LIN {X 0.250,Y -653.617,Z 434.422,A 0.000,B 0.000,C 90.000,E1 291.897} C_DIS
LIN {X 0.130,Y -656.048,Z 434.414,A 0.000,B 0.000,C 90.000,E1 290.429} C_DIS
LIN {X -0.023,Y -657.219,Z 434.410,A 0.000,B 0.000,C 90.000,E1 289.704} C_DIS
LIN {X -0.175,Y -658.743,Z 434.403,A 0.000,B 0.000,C 90.000,E1 288.489} C_DIS
LIN {X -0.311,Y -660.011,Z 434.396,A 0.000,B 0.000,C 90.000,E1 287.275} C_DIS
LIN {X 0.002,Y -660.962,Z 434.389,A 0.000,B 0.000,C 90.000,E1 286.024} C_DIS
LIN {X -0.211,Y -661.598,Z 434.384,A 0.000,B 0.000,C 90.000,E1 285.064} C_DIS
LIN {X -0.043,Y -662.268,Z 434.377,A 0.000,B 0.000,C 90.000,E1 283.828} C_DIS
LIN {X 0.046,Y -662.598,Z 434.369,A 0.000,B 0.000,C 90.000,E1 282.355} C_DIS
LIN {X 0.187,Y -662.630,Z 434.363,A 0.000,B 0.000,C 90.000,E1 281.366} C_DIS
LIN {X -0.196,Y -662.549,Z 434.358,A 0.000,B 0.000,C 90.000,E1 280.423} C_DIS
LIN {X -0.166,Y -662.206,Z 434.352,A 0.000,B 0.000,C 90.000,E1 279.443} C_DIS
LIN {X -0.133,Y -661.571,Z 434.346,A 0.000,B 0.000,C 90.000,E1 278.219} C_DIS
LIN {X -0.219,Y -660.695,Z 434.339,A 0.000,B 0.000,C 90.000,E1 277.004} C_DIS
LIN {X -0.202,Y -659.731,Z 434.333,A 0.000,B 0.000,C 90.000,E1 276.024} C_DIS
LIN {X 0.258,Y -658.178,Z 434.327,A 0.000,B 0.000,C 90.000,E1 274.759} C_DIS
LIN {X -0.012,Y -656.370,Z 434.320,A 0.000,B 0.000,C 90.000,E1 273.555} C_DIS
LIN {X 0.153,Y -653.762,Z 434.312,A 0.000,B 0.000,C 90.000,E1 272.064} C_DIS
LIN {X 0.225,Y -652.378,Z 434.307,A 0.000,B 0.000,C 90.000,E1 271.318} C_DIS
LIN {X -0.151,Y -649.780,Z 434.301,A 0.000,B 0.000,C 90.000,E1 270.115} C_DIS
LIN {X 0.082,Y -646.918,Z 434.294,A 0.000,B 0.000,C 90.000,E1 268.854} C_DIS
LIN {X 0.278,Y -643.759,Z 434.287,A 0.000,B 0.000,C 90.000,E1 267.593} C_DIS
LIN {X -0.217,Y -640.397,Z 434.280,A 0.000,B 0.000,C 90.000,E1 266.388} C_DIS
LIN {X 0.035,Y -635.593,Z 434.270,A 0.000,B 0.000,C 90.000,E1 264.609} C_DIS
LIN {X -0.274,Y -632.732,Z 434.265,A 0.000,B 0.000,C 90.000,E1 263.628} C_DIS
LIN {X 0.216,Y -628.308,Z 434.256,A 0.000,B 0.000,C 90.000,E1 262.064} C_DIS
LIN {X 0.217,Y -624.488,Z 434.249,A 0.000,B 0.000,C 90.000,E1 260.792} C_DIS
LIN {X -0.085,Y -619.805,Z 434.240,A 0.000,B 0.000,C 90.000,E1 259.285} C_DIS
LIN {X -0.012,Y -615.818,Z 434.233,A 0.000,B 0.000,C 90.000,E1 257.993} C_DIS
LIN {X 0.000,Y -611.688,Z 434.226,A 0.000,B 0.000,C 90.000,E1 256.700} C_DIS
LIN {X -0.062,Y -607.445,Z 434.219,A 0.000,B 0.000,C 90.000,E1 255.408} C_DIS
LIN {X -0.051,Y -603.009,Z 434.212,A 0.000,B 0.000,C 90.000,E1 254.102} C_DIS
LIN {X 0.164,Y -599.419,Z 434.206,A 0.000,B 0.000,C 90.000,E1 253.032} C_DIS
LIN {X 0.202,Y -594.834,Z 434.199,A 0.000,B 0.000,C 90.000,E1 251.710} C_DIS
LIN {X -0.204,Y -590.123,Z 434.191,A 0.000,B 0.000,C 90.000,E1 250.423} C_DIS
LIN {X -0.124,Y -585.262,Z 434.184,A 0.000,B 0.000,C 90.000,E1 249.082} C_DIS
LIN {X 0.080,Y -580.220,Z 434.176,A 0.000,B 0.000,C 90.000,E1 247.720} C_DIS
LIN {X -0.185,Y -576.063,Z 434.170,A 0.000,B 0.000,C 90.000,E1 246.666} C_DIS
LIN {X -0.079,Y -569.603,Z 434.161,A 0.000,B 0.000,C 90.000,E1 245.025} C_DIS
LIN {X 0.071,Y -564.128,Z 434.154,A 0.000,B 0.000,C 90.000,E1 243.640} C_DIS
LIN {X -0.133,Y -558.706,Z 434.146,A 0.000,B 0.000,C 90.000,E1 242.281} C_DIS
LIN {X -0.124,Y -551.162,Z 434.135,A 0.000,B 0.000,C 90.000,E1 240.333} C_DIS
LIN {X -0.258,Y -544.858,Z 434.126,A 0.000,B 0.000,C 90.000,E1 238.663} C_DIS
LIN {X 0.217,Y -538.693,Z 434.116,A 0.000,B 0.000,C 90.000,E1 236.914} C_DIS
LIN {X -0.047,Y -532.466,Z 434.107,A 0.000,B 0.000,C 90.000,E1 235.229} C_DIS
LIN {X -0.005,Y -526.440,Z 434.097,A 0.000,B 0.000,C 90.000,E1 233.497} C_DIS
LIN {X -0.174,Y -521.459,Z 434.089,A 0.000,B 0.000,C 90.000,E1 232.065} C_DIS
LIN {X -0.131,Y -509.297,Z 434.068,A 0.000,B 0.000,C 90.000,E1 228.243} C_DIS
LIN {X -0.002,Y -504.945,Z 434.060,A 0.000,B 0.000,C 90.000,E1 226.743} C_DIS
LIN {X -0.239,Y -499.025,Z 434.048,A 0.000,B 0.000,C 90.000,E1 224.676} C_DIS
LIN {X -0.110,Y -493.989,Z 434.038,A 0.000,B 0.000,C 90.000,E1 222.852} C_DIS
LIN {X 0.259,Y -489.097,Z 434.028,A 0.000,B 0.000,C 90.000,E1 220.987} C_DIS
LIN {X 0.200,Y -482.826,Z 434.014,A 0.000,B 0.000,C 90.000,E1 218.543} C_DIS
LIN {X 0.238,Y -477.527,Z 434.002,A 0.000,B 0.000,C 90.000,E1 216.377} C_DIS
LIN {X 0.237,Y -472.534,Z 433.990,A 0.000,B 0.000,C 90.000,E1 214.199} C_DIS
LIN {X 0.227,Y -467.724,Z 433.978,A 0.000,B 0.000,C 90.000,E1 212.005} C_DIS
LIN {X 0.092,Y -463.614,Z 433.967,A 0.000,B 0.000,C 90.000,E1 210.129} C_DIS
LIN {X 0.003,Y -460.931,Z 433.960,A 0.000,B 0.000,C 90.000,E1 208.871} C_DIS
LIN {X 0.172,Y -457.535,Z 433.952,A 0.000,B 0.000,C 90.000,E1 207.257} C_DIS
LIN {X 0.164,Y -453.407,Z 433.941,A 0.000,B 0.000,C 90.000,E1 205.335} C_DIS
LIN {X -0.203,Y -449.920,Z 433.932,A 0.000,B 0.000,C 90.000,E1 203.770} C_DIS
LIN {X 0.103,Y -445.038,Z 433.919,A 0.000,B 0.000,C 90.000,E1 201.461} C_DIS
LIN {X -0.102,Y -439.088,Z 433.903,A 0.000,B 0.000,C 90.000,E1 198.544} C_DIS
LIN {X 0.014,Y -435.531,Z 433.892,A 0.000,B 0.000,C 90.000,E1 196.551} C_DIS
LIN {X 0.213,Y -432.184,Z 433.881,A 0.000,B 0.000,C 90.000,E1 194.537} C_DIS
LIN {X -0.080,Y -428.469,Z 433.868,A 0.000,B 0.000,C 90.000,E1 192.243} C_DIS
LIN {X -0.141,Y -425.126,Z 433.855,A 0.000,B 0.000,C 90.000,E1 189.905} C_DIS
LIN {X -0.038,Y -422.611,Z 433.844,A 0.000,B 0.000,C 90.000,E1 187.871} C_DIS
LIN {X -0.093,Y -419.839,Z 433.831,A 0.000,B 0.000,C 90.000,E1 185.511} C_DIS
LIN {X -0.129,Y -416.249,Z 433.810,A 0.000,B 0.000,C 90.000,E1 181.776} C_DIS
LIN {X 0.004,Y -414.130,Z 433.793,A 0.000,B 0.000,C 90.000,E1 178.682} C_DIS
LIN {X 0.106,Y -412.775,Z 433.774,A 0.000,B 0.000,C 90.000,E1 175.241} C_DIS
LIN {X 0.048,Y -412.747,Z 433.747,A 0.000,B 0.000,C 90.000,E1 170.443} C_DIS
LIN {X -0.005,Y -413.462,Z 433.734,A 0.000,B 0.000,C 90.000,E1 168.049} C_DIS
LIN {X -0.003,Y -415.609,Z 433.713,A 0.000,B 0.000,C 90.000,E1 164.283} C_DIS
LIN {X -0.137,Y -418.945,Z 433.692,A 0.000,B 0.000,C 90.000,E1 160.550} C_DIS
LIN {X -0.099,Y -420.808,Z 433.682,A 0.000,B 0.000,C 90.000,E1 158.847} C_DIS
LIN {X -0.013,Y -424.715,Z 433.666,A 0.000,B 0.000,C 90.000,E1 155.793} C_DIS
LIN {X 0.191,Y -429.199,Z 433.649,A 0.000,B 0.000,C 90.000,E1 152.743} C_DIS
LIN {X -0.202,Y -433.759,Z 433.634,A 0.000,B 0.000,C 90.000,E1 150.127} C_DIS
LIN {X 0.018,Y -439.444,Z 433.617,A 0.000,B 0.000,C 90.000,E1 147.120} C_DIS
LIN {X 0.122,Y -444.910,Z 433.603,A 0.000,B 0.000,C 90.000,E1 144.482} C_DIS
LIN {X -0.009,Y -452.479,Z 433.585,A 0.000,B 0.000,C 90.000,E1 141.251} C_DIS
LIN {X -0.121,Y -458.108,Z 433.572,A 0.000,B 0.000,C 90.000,E1 139.013} C_DIS
LIN {X 0.047,Y -461.366,Z 433.565,A 0.000,B 0.000,C 90.000,E1 137.715} C_DIS
LIN {X -0.076,Y -464.446,Z 433.558,A 0.000,B 0.000,C 90.000,E1 136.458} C_DIS
LIN {X 0.174,Y -467.339,Z 433.551,A 0.000,B 0.000,C 90.000,E1 135.162} C_DIS
LIN {X -0.192,Y -469.929,Z 433.544,A 0.000,B 0.000,C 90.000,E1 133.947} C_DIS
LIN {X 0.051,Y -471.626,Z 433.539,A 0.000,B 0.000,C 90.000,E1 132.975} C_DIS
LIN {X -0.097,Y -472.687,Z 433.535,A 0.000,B 0.000,C 90.000,E1 132.366} C_DIS
LIN {X 0.301,Y -474.244,Z 433.528,A 0.000,B 0.000,C 90.000,E1 131.067} C_DIS
LIN {X -0.040,Y -474.992,Z 433.523,A 0.000,B 0.000,C 90.000,E1 130.172} C_DIS
LIN {X -0.159,Y -475.287,Z 433.520,A 0.000,B 0.000,C 90.000,E1 129.564} C_DIS
LIN {X 0.089,Y -475.389,Z 433.516,A 0.000,B 0.000,C 90.000,E1 128.910} C_DIS
LIN {X 0.133,Y -474.971,Z 433.511,A 0.000,B 0.000,C 90.000,E1 127.971} C_DIS
LIN {X -0.203,Y -474.105,Z 433.506,A 0.000,B 0.000,C 90.000,E1 127.076} C_DIS
LIN {X 0.203,Y -472.825,Z 433.501,A 0.000,B 0.000,C 90.000,E1 126.091} C_DIS
LIN {X -0.061,Y -471.250,Z 433.495,A 0.000,B 0.000,C 90.000,E1 125.185} C_DIS
LIN {X 0.151,Y -469.902,Z 433.492,A 0.000,B 0.000,C 90.000,E1 124.532} C_DIS
LIN {X -0.147,Y -467.559,Z 433.487,A 0.000,B 0.000,C 90.000,E1 123.627} C_DIS
LIN {X 0.160,Y -465.875,Z 433.483,A 0.000,B 0.000,C 90.000,E1 122.959} C_DIS
LIN {X -0.049,Y -462.004,Z 433.476,A 0.000,B 0.000,C 90.000,E1 121.720} C_DIS
LIN {X 0.106,Y -458.851,Z 433.471,A 0.000,B 0.000,C 90.000,E1 120.747} C_DIS
LIN {X 0.065,Y -455.443,Z 433.466,A 0.000,B 0.000,C 90.000,E1 119.795} C_DIS
LIN {X 0.243,Y -450.623,Z 433.458,A 0.000,B 0.000,C 90.000,E1 118.487} C_DIS
LIN {X 0.136,Y -445.682,Z 433.451,A 0.000,B 0.000,C 90.000,E1 117.206} C_DIS
LIN {X -0.021,Y -442.536,Z 433.447,A 0.000,B 0.000,C 90.000,E1 116.411} C_DIS
LIN {X 0.027,Y -441.320,Z 433.445,A 0.000,B 0.000,C 90.000,E1 116.104} C_DIS
LIN {X -0.013,Y -441.311,Z 433.445,A 0.000,B 0.000,C 90.000,E1 116.104} C_DIS
LIN {X -0.123,Y -444.764,Z 433.439,A 0.000,B 0.000,C 90.000,E1 114.951} C_DIS
LIN {X -0.153,Y -454.734,Z 433.415,A 0.000,B 0.000,C 90.000,E1 110.737} C_DIS
LIN {X -0.030,Y -457.370,Z 433.410,A 0.000,B 0.000,C 90.000,E1 109.758} C_DIS
LIN {X 0.055,Y -466.003,Z 433.387,A 0.000,B 0.000,C 90.000,E1 105.607} C_DIS
LIN {X -0.223,Y -467.570,Z 433.383,A 0.000,B 0.000,C 90.000,E1 105.009} C_DIS
LIN {X -0.040,Y -468.579,Z 433.380,A 0.000,B 0.000,C 90.000,E1 104.356} C_DIS
LIN {X 0.187,Y -475.803,Z 433.357,A 0.000,B 0.000,C 90.000,E1 100.254} C_DIS
LIN {X 0.026,Y -476.306,Z 433.355,A 0.000,B 0.000,C 90.000,E1 99.962} C_DIS
LIN {X -0.027,Y -481.790,Z 433.331,A 0.000,B 0.000,C 90.000,E1 95.625} C_DIS
LIN {X -0.180,Y -482.172,Z 433.330,A 0.000,B 0.000,C 90.000,E1 95.334} C_DIS
LIN {X 0.234,Y -485.309,Z 433.306,A 0.000,B 0.000,C 90.000,E1 90.974} C_DIS
LIN {X 0.059,Y -485.537,Z 433.304,A 0.000,B 0.000,C 90.000,E1 90.688} C_DIS
LIN {X -0.219,Y -486.320,Z 433.282,A 0.000,B 0.000,C 90.000,E1 86.731} C_DIS
LIN {X -0.084,Y -486.304,Z 433.278,A 0.000,B 0.000,C 90.000,E1 86.102} C_DIS
LIN {X 0.120,Y -484.696,Z 433.254,A 0.000,B 0.000,C 90.000,E1 81.781} C_DIS
LIN {X -0.011,Y -484.599,Z 433.253,A 0.000,B 0.000,C 90.000,E1 81.489} C_DIS
LIN {X -0.132,Y -480.533,Z 433.227,A 0.000,B 0.000,C 90.000,E1 76.881} C_DIS
LIN {X 0.232,Y -474.284,Z 433.201,A 0.000,B 0.000,C 90.000,E1 72.181} C_DIS
LIN {X 0.052,Y -473.846,Z 433.199,A 0.000,B 0.000,C 90.000,E1 71.891} C_DIS
LIN {X 0.160,Y -466.254,Z 433.175,A 0.000,B 0.000,C 90.000,E1 67.486} C_DIS
LIN {X 0.102,Y -465.824,Z 433.173,A 0.000,B 0.000,C 90.000,E1 67.177} C_DIS
LIN {X 0.194,Y -464.675,Z 433.170,A 0.000,B 0.000,C 90.000,E1 66.613} C_DIS
LIN {X -0.206,Y -464.561,Z 433.170,A 0.000,B 0.000,C 90.000,E1 66.613} C_DIS
LIN {X -0.246,Y -464.593,Z 433.170,A 0.000,B 0.000,C 90.000,E1 66.613} C_DIS
LIN {X -0.202,Y -470.674,Z 433.165,A 0.000,B 0.000,C 90.000,E1 65.793} C_DIS
LIN {X 0.072,Y -478.830,Z 433.159,A 0.000,B 0.000,C 90.000,E1 64.665} C_DIS
LIN {X 0.025,Y -487.955,Z 433.152,A 0.000,B 0.000,C 90.000,E1 63.435} C_DIS
LIN {X 0.069,Y -493.287,Z 433.148,A 0.000,B 0.000,C 90.000,E1 62.666} C_DIS
LIN {X -0.037,Y -499.111,Z 433.143,A 0.000,B 0.000,C 90.000,E1 61.769} C_DIS
LIN {X 0.050,Y -501.807,Z 433.141,A 0.000,B 0.000,C 90.000,E1 61.307} C_DIS
LIN {X -0.034,Y -505.087,Z 433.137,A 0.000,B 0.000,C 90.000,E1 60.717} C_DIS
LIN {X 0.048,Y -510.350,Z 433.132,A 0.000,B 0.000,C 90.000,E1 59.665} C_DIS
LIN {X -0.158,Y -513.474,Z 433.127,A 0.000,B 0.000,C 90.000,E1 58.948} C_DIS
LIN {X 0.102,Y -515.615,Z 433.124,A 0.000,B 0.000,C 90.000,E1 58.329} C_DIS
LIN {X 0.034,Y -518.068,Z 433.119,A 0.000,B 0.000,C 90.000,E1 57.454} C_DIS
LIN {X 0.336,Y -519.471,Z 433.116,A 0.000,B 0.000,C 90.000,E1 56.834} C_DIS
LIN {X -0.128,Y -520.943,Z 433.111,A 0.000,B 0.000,C 90.000,E1 56.008} C_DIS
LIN {X 0.198,Y -521.679,Z 433.108,A 0.000,B 0.000,C 90.000,E1 55.388} C_DIS
LIN {X 0.056,Y -522.345,Z 433.103,A 0.000,B 0.000,C 90.000,E1 54.529} C_DIS
LIN {X 0.038,Y -522.630,Z 433.098,A 0.000,B 0.000,C 90.000,E1 53.657} C_DIS
LIN {X 0.219,Y -522.554,Z 433.093,A 0.000,B 0.000,C 90.000,E1 52.763} C_DIS
LIN {X 0.088,Y -522.282,Z 433.088,A 0.000,B 0.000,C 90.000,E1 51.904} C_DIS
LIN {X 0.230,Y -521.477,Z 433.082,A 0.000,B 0.000,C 90.000,E1 50.723} C_DIS
LIN {X -0.039,Y -520.492,Z 433.076,A 0.000,B 0.000,C 90.000,E1 49.585} C_DIS
LIN {X 0.071,Y -519.255,Z 433.069,A 0.000,B 0.000,C 90.000,E1 48.405} C_DIS
LIN {X 0.115,Y -517.880,Z 433.063,A 0.000,B 0.000,C 90.000,E1 47.229} C_DIS
LIN {X -0.314,Y -516.077,Z 433.054,A 0.000,B 0.000,C 90.000,E1 45.810} C_DIS
LIN {X 0.115,Y -513.699,Z 433.043,A 0.000,B 0.000,C 90.000,E1 43.704} C_DIS
LIN {X -0.229,Y -511.495,Z 433.031,A 0.000,B 0.000,C 90.000,E1 41.676} C_DIS
LIN {X 0.133,Y -509.253,Z 433.020,A 0.000,B 0.000,C 90.000,E1 39.564} C_DIS
LIN {X -0.014,Y -507.725,Z 433.012,A 0.000,B 0.000,C 90.000,E1 38.096} C_DIS
LIN {X 0.210,Y -506.075,Z 433.003,A 0.000,B 0.000,C 90.000,E1 36.583} C_DIS
LIN {X -0.005,Y -503.988,Z 432.993,A 0.000,B 0.000,C 90.000,E1 34.818} C_DIS
LIN {X 0.261,Y -502.106,Z 432.985,A 0.000,B 0.000,C 90.000,E1 33.293} C_DIS
LIN {X -0.182,Y -499.737,Z 432.975,A 0.000,B 0.000,C 90.000,E1 31.544} C_DIS
LIN {X -0.241,Y -497.355,Z 432.965,A 0.000,B 0.000,C 90.000,E1 29.745} C_DIS
LIN {X 0.105,Y -494.576,Z 432.953,A 0.000,B 0.000,C 90.000,E1 27.590} C_DIS
LIN {X 0.176,Y -491.696,Z 432.940,A 0.000,B 0.000,C 90.000,E1 25.155} C_DIS
LIN {X -0.227,Y -488.994,Z 432.925,A 0.000,B 0.000,C 90.000,E1 22.461} C_DIS
LIN {X -0.029,Y -487.179,Z 432.911,A 0.000,B 0.000,C 90.000,E1 19.993} C_DIS
LIN {X -0.251,Y -485.990,Z 432.901,A 0.000,B 0.000,C 90.000,E1 18.181} C_DIS
LIN {X -0.040,Y -484.937,Z 432.892,A 0.000,B 0.000,C 90.000,E1 16.622} C_DIS
LIN {X -0.126,Y -483.398,Z 432.880,A 0.000,B 0.000,C 90.000,E1 14.481} C_DIS
LIN {X -0.043,Y -482.004,Z 432.867,A 0.000,B 0.000,C 90.000,E1 12.007} C_DIS
LIN {X -0.062,Y -481.145,Z 432.855,A 0.000,B 0.000,C 90.000,E1 9.849} C_DIS
LIN {X -0.184,Y -480.610,Z 432.843,A 0.000,B 0.000,C 90.000,E1 7.701} C_DIS
LIN {X -0.004,Y -480.570,Z 432.826,A 0.000,B 0.000,C 90.000,E1 4.588} C_DIS
LIN {X 0.000,Y -482.361,Z 432.800,A 0.000,B 0.000,C 90.000,E1 360.000} C_DIS
LIN {X 0.160,Y -485.658,Z 432.780,A 0.000,B 0.000,C 90.000,E1 356.388} C_DIS
LIN {X -0.125,Y -488.777,Z 432.766,A 0.000,B 0.000,C 90.000,E1 353.970} C_DIS
LIN {X -0.153,Y -491.901,Z 432.755,A 0.000,B 0.000,C 90.000,E1 351.837} C_DIS
LIN {X 0.130,Y -494.900,Z 432.744,A 0.000,B 0.000,C 90.000,E1 349.982} C_DIS
LIN {X -0.004,Y -498.684,Z 432.733,A 0.000,B 0.000,C 90.000,E1 347.881} C_DIS
LIN {X 0.050,Y -504.365,Z 432.718,A 0.000,B 0.000,C 90.000,E1 345.172} C_DIS
LIN {X 0.033,Y -509.308,Z 432.706,A 0.000,B 0.000,C 90.000,E1 343.087} C_DIS
LIN {X 0.050,Y -516.149,Z 432.691,A 0.000,B 0.000,C 90.000,E1 340.423} C_DIS
LIN {X 0.167,Y -521.709,Z 432.680,A 0.000,B 0.000,C 90.000,E1 338.358} C_DIS
LIN {X 0.152,Y -526.615,Z 432.670,A 0.000,B 0.000,C 90.000,E1 336.613} C_DIS
LIN {X 0.060,Y -530.634,Z 432.662,A 0.000,B 0.000,C 90.000,E1 335.177} C_DIS
LIN {X -0.024,Y -535.638,Z 432.653,A 0.000,B 0.000,C 90.000,E1 333.461} C_DIS
LIN {X -0.234,Y -540.608,Z 432.643,A 0.000,B 0.000,C 90.000,E1 331.769} C_DIS
LIN {X 0.153,Y -546.655,Z 432.632,A 0.000,B 0.000,C 90.000,E1 329.744} C_DIS
LIN {X 0.181,Y -550.009,Z 432.626,A 0.000,B 0.000,C 90.000,E1 328.614} C_DIS
LIN {X 0.081,Y -553.426,Z 432.620,A 0.000,B 0.000,C 90.000,E1 327.502} C_DIS
LIN {X 0.273,Y -557.520,Z 432.612,A 0.000,B 0.000,C 90.000,E1 326.087} C_DIS
LIN {X -0.077,Y -561.708,Z 432.604,A 0.000,B 0.000,C 90.000,E1 324.736} C_DIS
LIN {X -0.003,Y -567.630,Z 432.593,A 0.000,B 0.000,C 90.000,E1 322.798} C_DIS
LIN {X -0.181,Y -575.412,Z 432.580,A 0.000,B 0.000,C 90.000,E1 320.356} C_DIS
LIN {X -0.319,Y -579.884,Z 432.572,A 0.000,B 0.000,C 90.000,E1 319.013} C_DIS
LIN {X 0.001,Y -584.287,Z 432.565,A 0.000,B 0.000,C 90.000,E1 317.634} C_DIS
LIN {X 0.064,Y -591.385,Z 432.553,A 0.000,B 0.000,C 90.000,E1 315.486} C_DIS
LIN {X 0.124,Y -597.568,Z 432.542,A 0.000,B 0.000,C 90.000,E1 313.623} C_DIS
LIN {X 0.113,Y -602.918,Z 432.534,A 0.000,B 0.000,C 90.000,E1 312.043} C_DIS
LIN {X -0.005,Y -607.278,Z 432.526,A 0.000,B 0.000,C 90.000,E1 310.744} C_DIS
LIN {X 0.026,Y -611.536,Z 432.519,A 0.000,B 0.000,C 90.000,E1 309.439} C_DIS
LIN {X 0.230,Y -614.833,Z 432.513,A 0.000,B 0.000,C 90.000,E1 308.382} C_DIS
LIN {X -0.153,Y -619.620,Z 432.505,A 0.000,B 0.000,C 90.000,E1 306.870} C_DIS
LIN {X -0.273,Y -623.391,Z 432.498,A 0.000,B 0.000,C 90.000,E1 305.598} C_DIS
LIN {X 0.197,Y -626.396,Z 432.492,A 0.000,B 0.000,C 90.000,E1 304.532} C_DIS
LIN {X -0.164,Y -630.655,Z 432.484,A 0.000,B 0.000,C 90.000,E1 303.038} C_DIS
LIN {X 0.074,Y -634.037,Z 432.476,A 0.000,B 0.000,C 90.000,E1 301.750} C_DIS
LIN {X 0.000,Y -636.689,Z 432.471,A 0.000,B 0.000,C 90.000,E1 300.747} C_DIS
LIN {X 0.383,Y -640.443,Z 432.462,A 0.000,B 0.000,C 90.000,E1 299.205} C_DIS
LIN {X 0.141,Y -643.434,Z 432.456,A 0.000,B 0.000,C 90.000,E1 297.975} C_DIS
LIN {X -0.052,Y -646.266,Z 432.449,A 0.000,B 0.000,C 90.000,E1 296.744} C_DIS
LIN {X 0.375,Y -649.080,Z 432.442,A 0.000,B 0.000,C 90.000,E1 295.463} C_DIS
LIN {X -0.021,Y -651.658,Z 432.435,A 0.000,B 0.000,C 90.000,E1 294.259} C_DIS
LIN {X 0.058,Y -654.318,Z 432.427,A 0.000,B 0.000,C 90.000,E1 292.770} C_DIS
LIN {X 0.086,Y -656.437,Z 432.420,A 0.000,B 0.000,C 90.000,E1 291.535} C_DIS
LIN {X 0.148,Y -658.528,Z 432.413,A 0.000,B 0.000,C 90.000,E1 290.301} C_DIS
LIN {X 0.123,Y -659.895,Z 432.407,A 0.000,B 0.000,C 90.000,E1 289.322} C_DIS
LIN {X 0.005,Y -660.756,Z 432.403,A 0.000,B 0.000,C 90.000,E1 288.598} C_DIS
LIN {X -0.206,Y -661.850,Z 432.398,A 0.000,B 0.000,C 90.000,E1 287.638} C_DIS
LIN {X 0.233,Y -663.002,Z 432.390,A 0.000,B 0.000,C 90.000,E1 286.134} C_DIS
LIN {X -0.311,Y -663.823,Z 432.382,A 0.000,B 0.000,C 90.000,E1 284.717} C_DIS
LIN {X -0.012,Y -664.201,Z 432.376,A 0.000,B 0.000,C 90.000,E1 283.716} C_DIS
LIN {X 0.122,Y -664.502,Z 432.368,A 0.000,B 0.000,C 90.000,E1 282.243} C_DIS
LIN {X 0.333,Y -664.413,Z 432.361,A 0.000,B 0.000,C 90.000,E1 281.007} C_DIS
LIN {X -0.063,Y -664.332,Z 432.357,A 0.000,B 0.000,C 90.000,E1 280.310} C_DIS
LIN {X 0.197,Y -664.040,Z 432.353,A 0.000,B 0.000,C 90.000,E1 279.557} C_DIS
LIN {X 0.161,Y -663.393,Z 432.346,A 0.000,B 0.000,C 90.000,E1 278.341} C_DIS
LIN {X 0.114,Y -662.523,Z 432.340,A 0.000,B 0.000,C 90.000,E1 277.125} C_DIS
LIN {X 0.163,Y -661.604,Z 432.334,A 0.000,B 0.000,C 90.000,E1 276.144} C_DIS
LIN {X 0.008,Y -660.041,Z 432.327,A 0.000,B 0.000,C 90.000,E1 274.935} C_DIS
LIN {X -0.179,Y -658.276,Z 432.321,A 0.000,B 0.000,C 90.000,E1 273.726} C_DIS
LIN {X -0.248,Y -656.561,Z 432.315,A 0.000,B 0.000,C 90.000,E1 272.751} C_DIS
LIN {X 0.114,Y -654.384,Z 432.308,A 0.000,B 0.000,C 90.000,E1 271.489} C_DIS
LIN {X -0.231,Y -651.837,Z 432.302,A 0.000,B 0.000,C 90.000,E1 270.286} C_DIS
LIN {X -0.194,Y -650.159,Z 432.297,A 0.000,B 0.000,C 90.000,E1 269.542} C_DIS
LIN {X 0.257,Y -647.807,Z 432.292,A 0.000,B 0.000,C 90.000,E1 268.511} C_DIS
LIN {X -0.177,Y -644.600,Z 432.285,A 0.000,B 0.000,C 90.000,E1 267.306} C_DIS
LIN {X -0.021,Y -641.230,Z 432.278,A 0.000,B 0.000,C 90.000,E1 266.045} C_DIS
LIN {X 0.301,Y -636.462,Z 432.268,A 0.000,B 0.000,C 90.000,E1 264.261} C_DIS
LIN {X -0.269,Y -632.770,Z 432.261,A 0.000,B 0.000,C 90.000,E1 263.053} C_DIS
LIN {X -0.198,Y -629.042,Z 432.254,A 0.000,B 0.000,C 90.000,E1 261.781} C_DIS
LIN {X 0.209,Y -624.362,Z 432.246,A 0.000,B 0.000,C 90.000,E1 260.218} C_DIS
LIN {X -0.041,Y -621.256,Z 432.240,A 0.000,B 0.000,C 90.000,E1 259.218} C_DIS
LIN {X -0.062,Y -617.236,Z 432.233,A 0.000,B 0.000,C 90.000,E1 257.937} C_DIS
LIN {X 0.210,Y -613.952,Z 432.227,A 0.000,B 0.000,C 90.000,E1 256.881} C_DIS
LIN {X 0.084,Y -608.851,Z 432.219,A 0.000,B 0.000,C 90.000,E1 255.338} C_DIS
LIN {X 0.228,Y -605.294,Z 432.213,A 0.000,B 0.000,C 90.000,E1 254.283} C_DIS
LIN {X -0.206,Y -600.788,Z 432.206,A 0.000,B 0.000,C 90.000,E1 253.015} C_DIS
LIN {X -0.128,Y -596.175,Z 432.198,A 0.000,B 0.000,C 90.000,E1 251.692} C_DIS
LIN {X 0.302,Y -590.442,Z 432.189,A 0.000,B 0.000,C 90.000,E1 250.061} C_DIS
LIN {X -0.167,Y -585.534,Z 432.182,A 0.000,B 0.000,C 90.000,E1 248.773} C_DIS
LIN {X -0.226,Y -582.494,Z 432.178,A 0.000,B 0.000,C 90.000,E1 247.975} C_DIS
LIN {X -0.073,Y -577.287,Z 432.170,A 0.000,B 0.000,C 90.000,E1 246.613} C_DIS
LIN {X 0.211,Y -571.884,Z 432.163,A 0.000,B 0.000,C 90.000,E1 245.229} C_DIS
LIN {X -0.293,Y -565.305,Z 432.153,A 0.000,B 0.000,C 90.000,E1 243.640} C_DIS
LIN {X -0.178,Y -558.760,Z 432.144,A 0.000,B 0.000,C 90.000,E1 241.975} C_DIS
LIN {X 0.094,Y -551.235,Z 432.133,A 0.000,B 0.000,C 90.000,E1 239.999} C_DIS
LIN {X -0.008,Y -543.915,Z 432.122,A 0.000,B 0.000,C 90.000,E1 238.043} C_DIS
LIN {X -0.019,Y -538.781,Z 432.115,A 0.000,B 0.000,C 90.000,E1 236.628} C_DIS
LIN {X 0.159,Y -531.594,Z 432.104,A 0.000,B 0.000,C 90.000,E1 234.609} C_DIS
LIN {X -0.203,Y -527.621,Z 432.097,A 0.000,B 0.000,C 90.000,E1 233.497} C_DIS
LIN {X -0.066,Y -521.633,Z 432.087,A 0.000,B 0.000,C 90.000,E1 231.743} C_DIS
LIN {X -0.246,Y -510.451,Z 432.068,A 0.000,B 0.000,C 90.000,E1 228.243} C_DIS
LIN {X -0.094,Y -506.096,Z 432.060,A 0.000,B 0.000,C 90.000,E1 226.743} C_DIS
LIN {X 0.195,Y -501.012,Z 432.050,A 0.000,B 0.000,C 90.000,E1 224.919} C_DIS
LIN {X 0.003,Y -495.974,Z 432.040,A 0.000,B 0.000,C 90.000,E1 223.137} C_DIS
LIN {X 0.086,Y -491.067,Z 432.030,A 0.000,B 0.000,C 90.000,E1 221.310} C_DIS
LIN {X -0.282,Y -484.691,Z 432.016,A 0.000,B 0.000,C 90.000,E1 218.910} C_DIS
LIN {X -0.197,Y -480.868,Z 432.007,A 0.000,B 0.000,C 90.000,E1 217.363} C_DIS
LIN {X -0.098,Y -477.136,Z 431.999,A 0.000,B 0.000,C 90.000,E1 215.804} C_DIS
LIN {X -0.072,Y -473.599,Z 431.990,A 0.000,B 0.000,C 90.000,E1 214.246} C_DIS
LIN {X 0.173,Y -469.465,Z 431.980,A 0.000,B 0.000,C 90.000,E1 212.339} C_DIS
LIN {X 0.078,Y -465.324,Z 431.969,A 0.000,B 0.000,C 90.000,E1 210.463} C_DIS
LIN {X 0.016,Y -462.643,Z 431.962,A 0.000,B 0.000,C 90.000,E1 209.205} C_DIS
LIN {X -0.186,Y -459.232,Z 431.953,A 0.000,B 0.000,C 90.000,E1 207.641} C_DIS
LIN {X -0.152,Y -455.074,Z 431.943,A 0.000,B 0.000,C 90.000,E1 205.720} C_DIS
LIN {X 0.001,Y -450.847,Z 431.932,A 0.000,B 0.000,C 90.000,E1 203.770} C_DIS
LIN {X -0.121,Y -446.636,Z 431.921,A 0.000,B 0.000,C 90.000,E1 201.844} C_DIS
LIN {X -0.232,Y -441.821,Z 431.909,A 0.000,B 0.000,C 90.000,E1 199.577} C_DIS
LIN {X -0.208,Y -437.513,Z 431.896,A 0.000,B 0.000,C 90.000,E1 197.275} C_DIS
LIN {X 0.160,Y -434.104,Z 431.885,A 0.000,B 0.000,C 90.000,E1 195.245} C_DIS
LIN {X -0.195,Y -430.842,Z 431.874,A 0.000,B 0.000,C 90.000,E1 193.300} C_DIS
LIN {X 0.091,Y -426.347,Z 431.857,A 0.000,B 0.000,C 90.000,E1 190.254} C_DIS
LIN {X -0.172,Y -423.339,Z 431.844,A 0.000,B 0.000,C 90.000,E1 187.936} C_DIS
LIN {X -0.150,Y -420.537,Z 431.831,A 0.000,B 0.000,C 90.000,E1 185.568} C_DIS
LIN {X 0.134,Y -418.082,Z 431.818,A 0.000,B 0.000,C 90.000,E1 183.154} C_DIS
LIN {X -0.115,Y -416.380,Z 431.806,A 0.000,B 0.000,C 90.000,E1 181.146} C_DIS
LIN {X 0.014,Y -414.582,Z 431.791,A 0.000,B 0.000,C 90.000,E1 178.396} C_DIS
LIN {X 0.165,Y -413.336,Z 431.772,A 0.000,B 0.000,C 90.000,E1 174.951} C_DIS
LIN {X 0.072,Y -413.321,Z 431.749,A 0.000,B 0.000,C 90.000,E1 170.849} C_DIS
LIN {X -0.004,Y -414.086,Z 431.734,A 0.000,B 0.000,C 90.000,E1 168.117} C_DIS
LIN {X -0.133,Y -416.463,Z 431.711,A 0.000,B 0.000,C 90.000,E1 164.031} C_DIS
LIN {X 0.019,Y -419.550,Z 431.692,A 0.000,B 0.000,C 90.000,E1 160.604} C_DIS
LIN {X -0.145,Y -421.846,Z 431.681,A 0.000,B 0.000,C 90.000,E1 158.592} C_DIS
LIN {X -0.015,Y -425.813,Z 431.664,A 0.000,B 0.000,C 90.000,E1 155.537} C_DIS
LIN {X -0.150,Y -430.406,Z 431.647,A 0.000,B 0.000,C 90.000,E1 152.538} C_DIS
LIN {X -0.126,Y -435.058,Z 431.633,A 0.000,B 0.000,C 90.000,E1 149.871} C_DIS
LIN {X -0.236,Y -440.907,Z 431.616,A 0.000,B 0.000,C 90.000,E1 146.914} C_DIS
LIN {X -0.088,Y -446.508,Z 431.602,A 0.000,B 0.000,C 90.000,E1 144.276} C_DIS
LIN {X 0.121,Y -454.275,Z 431.584,A 0.000,B 0.000,C 90.000,E1 141.009} C_DIS
LIN {X 0.067,Y -460.063,Z 431.571,A 0.000,B 0.000,C 90.000,E1 138.771} C_DIS
LIN {X 0.270,Y -463.343,Z 431.564,A 0.000,B 0.000,C 90.000,E1 137.472} C_DIS
LIN {X 0.182,Y -466.478,Z 431.557,A 0.000,B 0.000,C 90.000,E1 136.215} C_DIS
LIN {X -0.198,Y -469.341,Z 431.550,A 0.000,B 0.000,C 90.000,E1 135.000} C_DIS
LIN {X 0.044,Y -471.321,Z 431.545,A 0.000,B 0.000,C 90.000,E1 134.028} C_DIS
LIN {X -0.017,Y -473.182,Z 431.539,A 0.000,B 0.000,C 90.000,E1 133.095} C_DIS
LIN {X -0.054,Y -474.716,Z 431.534,A 0.000,B 0.000,C 90.000,E1 132.162} C_DIS
LIN {X 0.023,Y -476.284,Z 431.527,A 0.000,B 0.000,C 90.000,E1 130.906} C_DIS
LIN {X 0.168,Y -477.141,Z 431.520,A 0.000,B 0.000,C 90.000,E1 129.644} C_DIS
LIN {X -0.142,Y -477.272,Z 431.515,A 0.000,B 0.000,C 90.000,E1 128.749} C_DIS
LIN {X -0.079,Y -476.803,Z 431.510,A 0.000,B 0.000,C 90.000,E1 127.810} C_DIS
LIN {X -0.019,Y -475.852,Z 431.505,A 0.000,B 0.000,C 90.000,E1 126.870} C_DIS
LIN {X 0.027,Y -474.566,Z 431.500,A 0.000,B 0.000,C 90.000,E1 125.931} C_DIS
LIN {X -0.008,Y -473.542,Z 431.496,A 0.000,B 0.000,C 90.000,E1 125.311} C_DIS
LIN {X -0.047,Y -472.245,Z 431.493,A 0.000,B 0.000,C 90.000,E1 124.692} C_DIS
LIN {X -0.315,Y -469.970,Z 431.488,A 0.000,B 0.000,C 90.000,E1 123.785} C_DIS
LIN {X 0.036,Y -467.386,Z 431.482,A 0.000,B 0.000,C 90.000,E1 122.801} C_DIS
LIN {X -0.004,Y -463.477,Z 431.475,A 0.000,B 0.000,C 90.000,E1 121.544} C_DIS
LIN {X 0.012,Y -460.246,Z 431.470,A 0.000,B 0.000,C 90.000,E1 120.590} C_DIS
LIN {X 0.154,Y -456.775,Z 431.465,A 0.000,B 0.000,C 90.000,E1 119.617} C_DIS
LIN {X 0.097,Y -451.218,Z 431.457,A 0.000,B 0.000,C 90.000,E1 118.180} C_DIS
LIN {X 0.062,Y -444.893,Z 431.448,A 0.000,B 0.000,C 90.000,E1 116.565} C_DIS
LIN {X 0.092,Y -442.016,Z 431.444,A 0.000,B 0.000,C 90.000,E1 115.848} C_DIS
LIN {X 0.052,Y -442.026,Z 431.444,A 0.000,B 0.000,C 90.000,E1 115.848} C_DIS
LIN {X 0.179,Y -444.263,Z 431.440,A 0.000,B 0.000,C 90.000,E1 115.079} C_DIS
LIN {X 0.033,Y -445.119,Z 431.438,A 0.000,B 0.000,C 90.000,E1 114.771} C_DIS
LIN {X 0.140,Y -454.290,Z 431.416,A 0.000,B 0.000,C 90.000,E1 110.865} C_DIS
LIN {X -0.168,Y -456.956,Z 431.411,A 0.000,B 0.000,C 90.000,E1 109.939} C_DIS
LIN {X 0.070,Y -458.227,Z 431.407,A 0.000,B 0.000,C 90.000,E1 109.268} C_DIS
LIN {X -0.181,Y -466.381,Z 431.386,A 0.000,B 0.000,C 90.000,E1 105.481} C_DIS
LIN {X -0.008,Y -467.902,Z 431.382,A 0.000,B 0.000,C 90.000,E1 104.828} C_DIS
LIN {X 0.020,Y -475.471,Z 431.358,A 0.000,B 0.000,C 90.000,E1 100.433} C_DIS
LIN {X -0.142,Y -476.116,Z 431.356,A 0.000,B 0.000,C 90.000,E1 100.141} C_DIS
LIN {X 0.142,Y -482.034,Z 431.330,A 0.000,B 0.000,C 90.000,E1 95.454} C_DIS
LIN {X -0.068,Y -485.470,Z 431.305,A 0.000,B 0.000,C 90.000,E1 90.859} C_DIS
LIN {X 0.035,Y -485.536,Z 431.296,A 0.000,B 0.000,C 90.000,E1 89.312} C_DIS
LIN {X -0.035,Y -486.385,Z 431.281,A 0.000,B 0.000,C 90.000,E1 86.560} C_DIS
LIN {X -0.210,Y -486.364,Z 431.279,A 0.000,B 0.000,C 90.000,E1 86.274} C_DIS
LIN {X -0.122,Y -484.690,Z 431.254,A 0.000,B 0.000,C 90.000,E1 81.659} C_DIS
LIN {X -0.107,Y -483.701,Z 431.249,A 0.000,B 0.000,C 90.000,E1 80.735} C_DIS
LIN {X 0.256,Y -480.629,Z 431.228,A 0.000,B 0.000,C 90.000,E1 76.992} C_DIS
LIN {X 0.115,Y -480.313,Z 431.226,A 0.000,B 0.000,C 90.000,E1 76.700} C_DIS
LIN {X 0.018,Y -474.130,Z 431.200,A 0.000,B 0.000,C 90.000,E1 72.054} C_DIS
LIN {X -0.114,Y -465.599,Z 431.172,A 0.000,B 0.000,C 90.000,E1 67.050} C_DIS
LIN {X 0.079,Y -465.065,Z 431.171,A 0.000,B 0.000,C 90.000,E1 66.794} C_DIS
LIN {X 0.039,Y -465.074,Z 431.171,A 0.000,B 0.000,C 90.000,E1 66.794} C_DIS
LIN {X 0.079,Y -471.544,Z 431.166,A 0.000,B 0.000,C 90.000,E1 65.921} C_DIS
LIN {X -0.041,Y -479.709,Z 431.160,A 0.000,B 0.000,C 90.000,E1 64.845} C_DIS
LIN {X -0.067,Y -489.968,Z 431.153,A 0.000,B 0.000,C 90.000,E1 63.461} C_DIS
LIN {X -0.011,Y -495.214,Z 431.148,A 0.000,B 0.000,C 90.000,E1 62.692} C_DIS
LIN {X -0.149,Y -499.110,Z 431.145,A 0.000,B 0.000,C 90.000,E1 62.103} C_DIS
LIN {X -0.061,Y -501.930,Z 431.142,A 0.000,B 0.000,C 90.000,E1 61.641} C_DIS
LIN {X 0.104,Y -506.112,Z 431.138,A 0.000,B 0.000,C 90.000,E1 60.873} C_DIS
LIN {X -0.247,Y -511.354,Z 431.133,A 0.000,B 0.000,C 90.000,E1 59.871} C_DIS
LIN {X -0.183,Y -514.587,Z 431.128,A 0.000,B 0.000,C 90.000,E1 59.125} C_DIS
LIN {X -0.180,Y -516.717,Z 431.125,A 0.000,B 0.000,C 90.000,E1 58.535} C_DIS
LIN {X -0.239,Y -519.291,Z 431.120,A 0.000,B 0.000,C 90.000,E1 57.661} C_DIS
LIN {X 0.071,Y -520.692,Z 431.117,A 0.000,B 0.000,C 90.000,E1 57.041} C_DIS
LIN {X 0.053,Y -522.269,Z 431.112,A 0.000,B 0.000,C 90.000,E1 56.167} C_DIS
LIN {X -0.090,Y -523.292,Z 431.107,A 0.000,B 0.000,C 90.000,E1 55.308} C_DIS
LIN {X 0.254,Y -523.732,Z 431.104,A 0.000,B 0.000,C 90.000,E1 54.689} C_DIS
LIN {X 0.136,Y -524.053,Z 431.099,A 0.000,B 0.000,C 90.000,E1 53.829} C_DIS
LIN {X -0.013,Y -523.903,Z 431.093,A 0.000,B 0.000,C 90.000,E1 52.683} C_DIS
LIN {X -0.128,Y -523.557,Z 431.088,A 0.000,B 0.000,C 90.000,E1 51.823} C_DIS
LIN {X 0.036,Y -522.709,Z 431.081,A 0.000,B 0.000,C 90.000,E1 50.642} C_DIS
LIN {X 0.183,Y -521.654,Z 431.075,A 0.000,B 0.000,C 90.000,E1 49.461} C_DIS
LIN {X -0.085,Y -520.373,Z 431.068,A 0.000,B 0.000,C 90.000,E1 48.324} C_DIS
LIN {X -0.022,Y -518.952,Z 431.062,A 0.000,B 0.000,C 90.000,E1 47.148} C_DIS
LIN {X 0.122,Y -516.363,Z 431.051,A 0.000,B 0.000,C 90.000,E1 45.081} C_DIS
LIN {X 0.201,Y -513.998,Z 431.039,A 0.000,B 0.000,C 90.000,E1 43.014} C_DIS
LIN {X 0.084,Y -512.406,Z 431.031,A 0.000,B 0.000,C 90.000,E1 41.553} C_DIS
LIN {X 0.086,Y -510.192,Z 431.019,A 0.000,B 0.000,C 90.000,E1 39.483} C_DIS
LIN {X -0.046,Y -508.631,Z 431.011,A 0.000,B 0.000,C 90.000,E1 38.016} C_DIS
LIN {X 0.094,Y -506.576,Z 431.001,A 0.000,B 0.000,C 90.000,E1 36.217} C_DIS
LIN {X -0.008,Y -504.818,Z 430.993,A 0.000,B 0.000,C 90.000,E1 34.739} C_DIS
LIN {X -0.312,Y -503.309,Z 430.986,A 0.000,B 0.000,C 90.000,E1 33.579} C_DIS
LIN {X -0.031,Y -500.942,Z 430.976,A 0.000,B 0.000,C 90.000,E1 31.750} C_DIS
LIN {X 0.188,Y -498.567,Z 430.966,A 0.000,B 0.000,C 90.000,E1 29.922} C_DIS
LIN {X -0.116,Y -495.785,Z 430.955,A 0.000,B 0.000,C 90.000,E1 27.847} C_DIS
LIN {X 0.240,Y -492.550,Z 430.940,A 0.000,B 0.000,C 90.000,E1 25.079} C_DIS
LIN {X -0.117,Y -489.576,Z 430.923,A 0.000,B 0.000,C 90.000,E1 22.078} C_DIS
LIN {X -0.102,Y -488.044,Z 430.911,A 0.000,B 0.000,C 90.000,E1 19.939} C_DIS
LIN {X -0.148,Y -486.832,Z 430.901,A 0.000,B 0.000,C 90.000,E1 18.109} C_DIS
LIN {X 0.070,Y -485.784,Z 430.892,A 0.000,B 0.000,C 90.000,E1 16.551} C_DIS
LIN {X -0.006,Y -484.224,Z 430.880,A 0.000,B 0.000,C 90.000,E1 14.411} C_DIS
LIN {X -0.014,Y -482.876,Z 430.866,A 0.000,B 0.000,C 90.000,E1 11.951} C_DIS
LIN {X 0.214,Y -482.124,Z 430.856,A 0.000,B 0.000,C 90.000,E1 10.074} C_DIS
LIN {X 0.040,Y -481.572,Z 430.844,A 0.000,B 0.000,C 90.000,E1 7.936} C_DIS
LIN {X 0.115,Y -481.473,Z 430.825,A 0.000,B 0.000,C 90.000,E1 4.531} C_DIS
LIN {X -0.152,Y -482.753,Z 430.805,A 0.000,B 0.000,C 90.000,E1 0.859} C_DIS
LIN {X 0.023,Y -486.974,Z 430.778,A 0.000,B 0.000,C 90.000,E1 356.102} C_DIS
LIN {X -0.231,Y -490.167,Z 430.765,A 0.000,B 0.000,C 90.000,E1 353.685} C_DIS
LIN {X -0.057,Y -492.915,Z 430.755,A 0.000,B 0.000,C 90.000,E1 351.837} C_DIS
LIN {X 0.159,Y -496.450,Z 430.743,A 0.000,B 0.000,C 90.000,E1 349.690} C_DIS
LIN {X -0.126,Y -504.119,Z 430.721,A 0.000,B 0.000,C 90.000,E1 345.811} C_DIS
LIN {X -0.241,Y -510.389,Z 430.706,A 0.000,B 0.000,C 90.000,E1 343.142} C_DIS
LIN {X 0.175,Y -516.426,Z 430.693,A 0.000,B 0.000,C 90.000,E1 340.732} C_DIS
LIN {X 0.193,Y -520.376,Z 430.685,A 0.000,B 0.000,C 90.000,E1 339.263} C_DIS
LIN {X 0.123,Y -526.067,Z 430.674,A 0.000,B 0.000,C 90.000,E1 337.230} C_DIS
LIN {X 0.027,Y -530.139,Z 430.666,A 0.000,B 0.000,C 90.000,E1 335.793} C_DIS
LIN {X -0.143,Y -536.776,Z 430.653,A 0.000,B 0.000,C 90.000,E1 333.512} C_DIS
LIN {X 0.156,Y -541.787,Z 430.643,A 0.000,B 0.000,C 90.000,E1 331.769} C_DIS
LIN {X 0.105,Y -547.854,Z 430.632,A 0.000,B 0.000,C 90.000,E1 329.793} C_DIS
LIN {X 0.155,Y -551.280,Z 430.626,A 0.000,B 0.000,C 90.000,E1 328.663} C_DIS
LIN {X 0.312,Y -555.531,Z 430.618,A 0.000,B 0.000,C 90.000,E1 327.248} C_DIS
LIN {X 0.072,Y -559.666,Z 430.611,A 0.000,B 0.000,C 90.000,E1 325.881} C_DIS
LIN {X 0.219,Y -563.894,Z 430.603,A 0.000,B 0.000,C 90.000,E1 324.482} C_DIS
LIN {X 0.102,Y -568.988,Z 430.594,A 0.000,B 0.000,C 90.000,E1 322.844} C_DIS
LIN {X -0.015,Y -576.822,Z 430.580,A 0.000,B 0.000,C 90.000,E1 320.400} C_DIS
LIN {X 0.045,Y -582.193,Z 430.571,A 0.000,B 0.000,C 90.000,E1 318.771} C_DIS
LIN {X 0.156,Y -587.490,Z 430.562,A 0.000,B 0.000,C 90.000,E1 317.148} C_DIS
LIN {X -0.054,Y -592.853,Z 430.553,A 0.000,B 0.000,C 90.000,E1 315.567} C_DIS
LIN {X 0.259,Y -598.200,Z 430.544,A 0.000,B 0.000,C 90.000,E1 313.947} C_DIS
LIN {X -0.377,Y -602.670,Z 430.537,A 0.000,B 0.000,C 90.000,E1 312.690} C_DIS
LIN {X 0.107,Y -606.237,Z 430.531,A 0.000,B 0.000,C 90.000,E1 311.595} C_DIS
LIN {X 0.047,Y -610.577,Z 430.524,A 0.000,B 0.000,C 90.000,E1 310.297} C_DIS
LIN {X -0.043,Y -615.674,Z 430.515,A 0.000,B 0.000,C 90.000,E1 308.749} C_DIS
LIN {X -0.035,Y -620.519,Z 430.507,A 0.000,B 0.000,C 90.000,E1 307.202} C_DIS
LIN {X -0.148,Y -624.346,Z 430.500,A 0.000,B 0.000,C 90.000,E1 305.931} C_DIS
LIN {X 0.320,Y -628.106,Z 430.492,A 0.000,B 0.000,C 90.000,E1 304.612} C_DIS
LIN {X 0.343,Y -632.386,Z 430.484,A 0.000,B 0.000,C 90.000,E1 303.086} C_DIS
LIN {X 0.239,Y -635.145,Z 430.478,A 0.000,B 0.000,C 90.000,E1 302.084} C_DIS
LIN {X 0.004,Y -638.511,Z 430.471,A 0.000,B 0.000,C 90.000,E1 300.846} C_DIS
LIN {X 0.095,Y -642.293,Z 430.463,A 0.000,B 0.000,C 90.000,E1 299.333} C_DIS
LIN {X -0.120,Y -645.328,Z 430.456,A 0.000,B 0.000,C 90.000,E1 298.103} C_DIS
LIN {X -0.196,Y -648.731,Z 430.448,A 0.000,B 0.000,C 90.000,E1 296.616} C_DIS
LIN {X 0.272,Y -651.506,Z 430.441,A 0.000,B 0.000,C 90.000,E1 295.335} C_DIS
LIN {X -0.088,Y -654.027,Z 430.434,A 0.000,B 0.000,C 90.000,E1 294.131} C_DIS
LIN {X 0.037,Y -656.715,Z 430.426,A 0.000,B 0.000,C 90.000,E1 292.642} C_DIS
LIN {X 0.103,Y -658.852,Z 430.419,A 0.000,B 0.000,C 90.000,E1 291.408} C_DIS
LIN {X 0.087,Y -660.569,Z 430.414,A 0.000,B 0.000,C 90.000,E1 290.429} C_DIS
LIN {X -0.014,Y -662.217,Z 430.407,A 0.000,B 0.000,C 90.000,E1 289.214} C_DIS
LIN {X -0.090,Y -663.547,Z 430.400,A 0.000,B 0.000,C 90.000,E1 288.000} C_DIS
LIN {X -0.251,Y -664.842,Z 430.392,A 0.000,B 0.000,C 90.000,E1 286.551} C_DIS
LIN {X -0.030,Y -665.752,Z 430.382,A 0.000,B 0.000,C 90.000,E1 284.828} C_DIS
LIN {X 0.206,Y -666.034,Z 430.376,A 0.000,B 0.000,C 90.000,E1 283.592} C_DIS
LIN {X -0.201,Y -666.158,Z 430.369,A 0.000,B 0.000,C 90.000,E1 282.411} C_DIS
LIN {X -0.016,Y -666.090,Z 430.363,A 0.000,B 0.000,C 90.000,E1 281.422} C_DIS
LIN {X 0.092,Y -665.817,Z 430.357,A 0.000,B 0.000,C 90.000,E1 280.197} C_DIS
LIN {X 0.281,Y -665.304,Z 430.351,A 0.000,B 0.000,C 90.000,E1 279.208} C_DIS
LIN {X 0.264,Y -664.518,Z 430.345,A 0.000,B 0.000,C 90.000,E1 277.992} C_DIS
LIN {X -0.319,Y -663.797,Z 430.339,A 0.000,B 0.000,C 90.000,E1 277.068} C_DIS
LIN {X -0.251,Y -662.825,Z 430.334,A 0.000,B 0.000,C 90.000,E1 276.087} C_DIS
LIN {X 0.274,Y -661.280,Z 430.327,A 0.000,B 0.000,C 90.000,E1 274.821} C_DIS
LIN {X 0.108,Y -659.551,Z 430.320,A 0.000,B 0.000,C 90.000,E1 273.612} C_DIS
LIN {X -0.133,Y -657.423,Z 430.313,A 0.000,B 0.000,C 90.000,E1 272.407} C_DIS
LIN {X -0.217,Y -655.674,Z 430.308,A 0.000,B 0.000,C 90.000,E1 271.432} C_DIS
LIN {X 0.313,Y -653.708,Z 430.302,A 0.000,B 0.000,C 90.000,E1 270.401} C_DIS
LIN {X 0.164,Y -651.550,Z 430.297,A 0.000,B 0.000,C 90.000,E1 269.427} C_DIS
END
